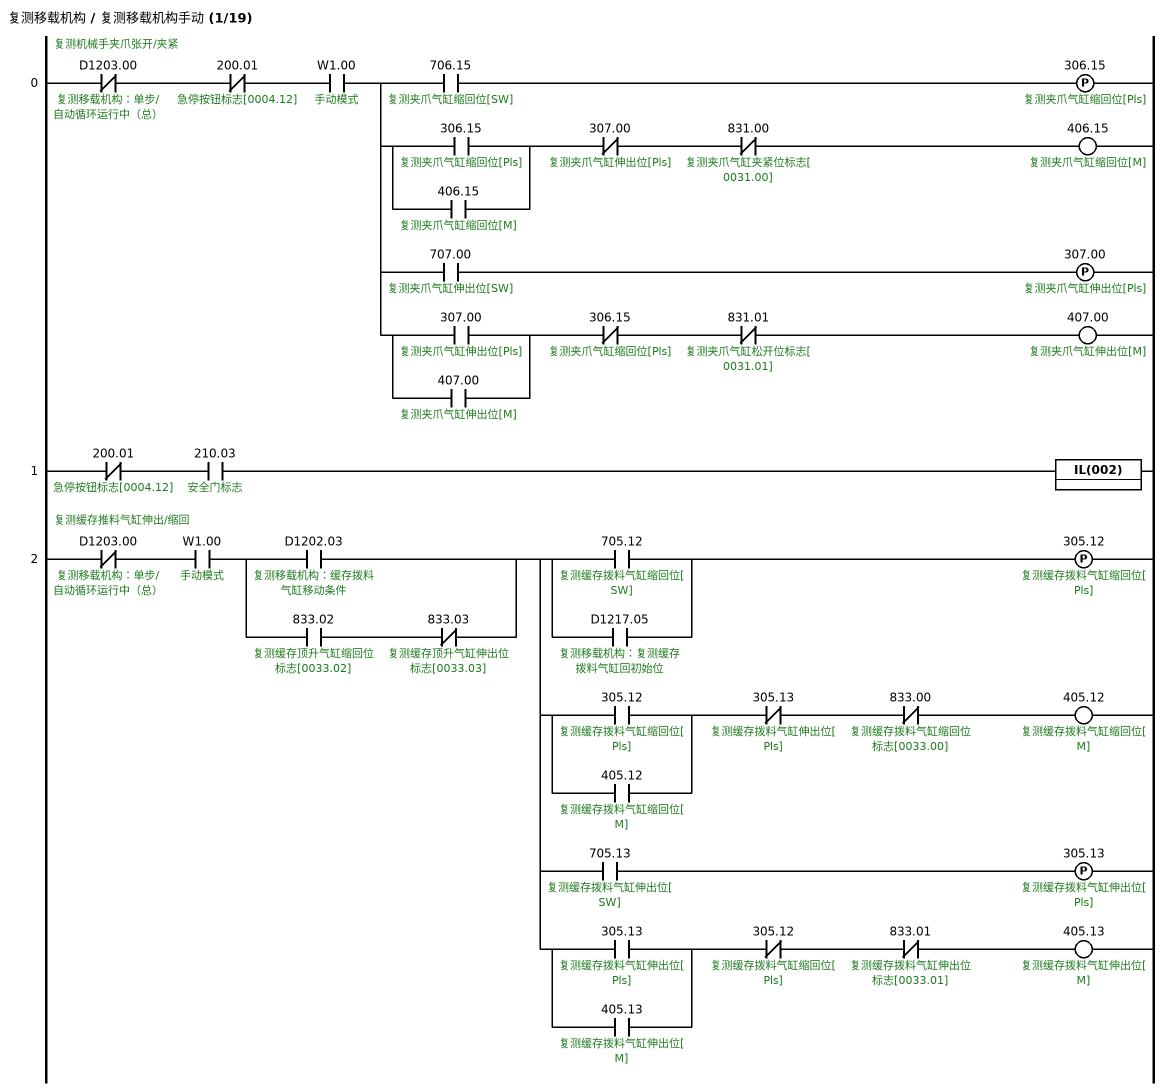
; [picture p552: 复测移载机构 / 复测移载机构手动, rungs 0-2]
; rung 0: 复测机械手夹爪张开/夹紧
LDNOT D1203.00  ; 复测移载机构：单步/自动循环运行中（总）
ANDNOT 200.01  ; 急停按钮标志[0004.12]
AND W1.00  ; 手动模式
OUT TR0
AND 706.15  ; 复测夹爪气缸缩回位[SW]
DIFU(013) 306.15  ; 复测夹爪气缸缩回位[Pls]
LD TR0
LD 306.15  ; 复测夹爪气缸缩回位[Pls]
OR 406.15  ; 复测夹爪气缸缩回位[M]
ANDLD
ANDNOT 307.00  ; 复测夹爪气缸伸出位[Pls]
ANDNOT 831.00  ; 复测夹爪气缸夹紧位标志[0031.00]
OUT 406.15  ; 复测夹爪气缸缩回位[M]
LD TR0
AND 707.00  ; 复测夹爪气缸伸出位[SW]
DIFU(013) 307.00  ; 复测夹爪气缸伸出位[Pls]
LD TR0
LD 307.00  ; 复测夹爪气缸伸出位[Pls]
OR 407.00  ; 复测夹爪气缸伸出位[M]
ANDLD
ANDNOT 306.15  ; 复测夹爪气缸缩回位[Pls]
ANDNOT 831.01  ; 复测夹爪气缸松开位标志[0031.01]
OUT 407.00  ; 复测夹爪气缸伸出位[M]
; rung 1
LDNOT 200.01  ; 急停按钮标志[0004.12]
AND 210.03  ; 安全门标志
IL(002)
; rung 2: 复测缓存推料气缸伸出/缩回
LDNOT D1203.00  ; 复测移载机构：单步/自动循环运行中（总）
AND W1.00  ; 手动模式
LD D1202.03  ; 复测移载机构：缓存拨料气缸移动条件
LD 833.02  ; 复测缓存顶升气缸缩回位标志[0033.02]
ANDNOT 833.03  ; 复测缓存顶升气缸伸出位标志[0033.03]
ORLD
ANDLD
OUT TR0
LD 705.12  ; 复测缓存拨料气缸缩回位[SW]
OR D1217.05  ; 复测移载机构：复测缓存拨料气缸回初始位
ANDLD
DIFU(013) 305.12  ; 复测缓存拨料气缸缩回位[Pls]
LD TR0
LD 305.12  ; 复测缓存拨料气缸缩回位[Pls]
OR 405.12  ; 复测缓存拨料气缸缩回位[M]
ANDLD
ANDNOT 305.13  ; 复测缓存拨料气缸伸出位[Pls]
ANDNOT 833.00  ; 复测缓存拨料气缸缩回位标志[0033.00]
OUT 405.12  ; 复测缓存拨料气缸缩回位[M]
LD TR0
AND 705.13  ; 复测缓存拨料气缸伸出位[SW]
DIFU(013) 305.13  ; 复测缓存拨料气缸伸出位[Pls]
LD TR0
LD 305.13  ; 复测缓存拨料气缸伸出位[Pls]
OR 405.13  ; 复测缓存拨料气缸伸出位[M]
ANDLD
ANDNOT 305.12  ; 复测缓存拨料气缸缩回位[Pls]
ANDNOT 833.01  ; 复测缓存拨料气缸伸出位标志[0033.01]
OUT 405.13  ; 复测缓存拨料气缸伸出位[M]

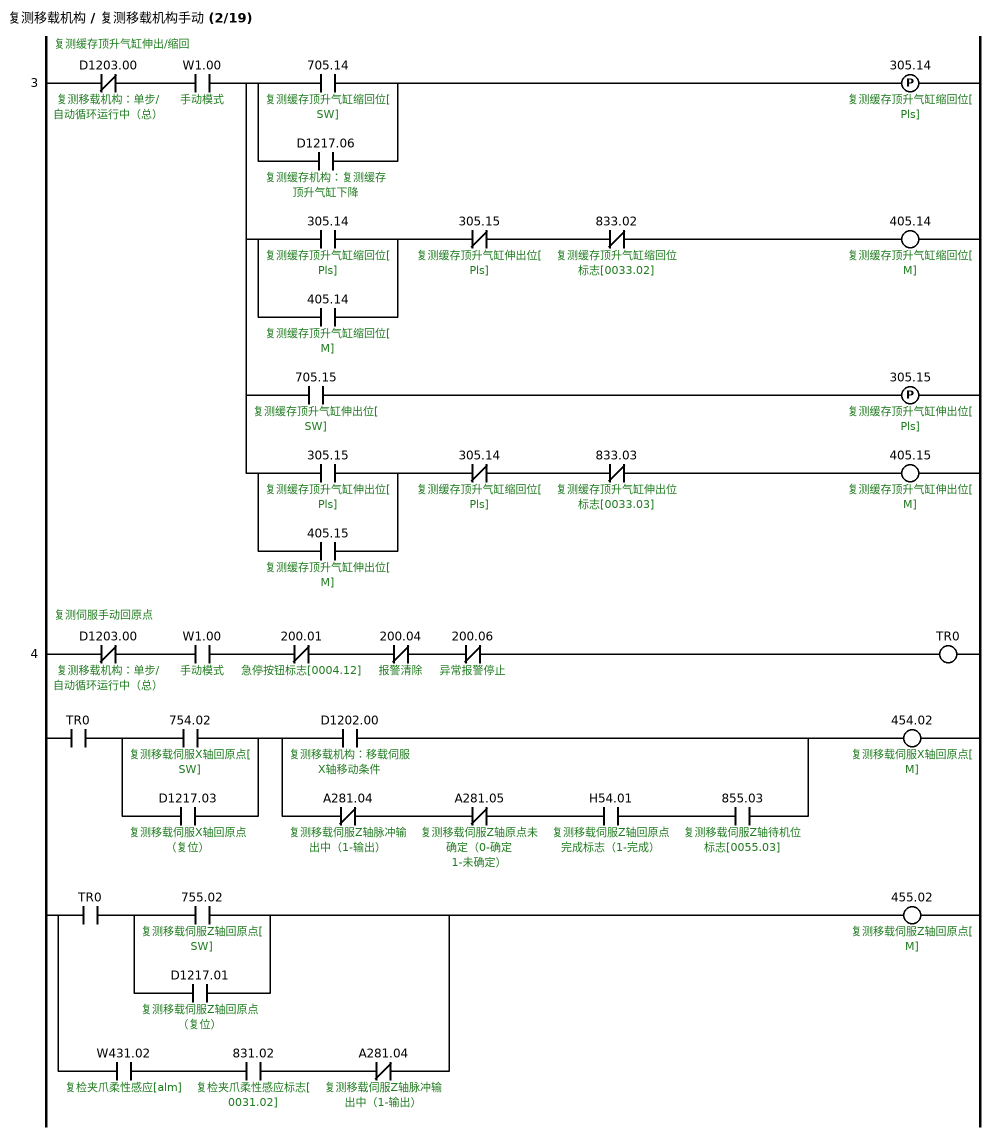
; rung 3: 复测缓存顶升气缸伸出/缩回
LDNOT D1203.00  ; 复测移载机构：单步/自动循环运行中（总）
AND W1.00  ; 手动模式
OUT TR0
LD 705.14  ; 复测缓存顶升气缸缩回位[SW]
OR D1217.06  ; 复测缓存机构：复测缓存顶升气缸下降
ANDLD
DIFU(013) 305.14  ; 复测缓存顶升气缸缩回位[Pls]
LD TR0
LD 305.14  ; 复测缓存顶升气缸缩回位[Pls]
OR 405.14  ; 复测缓存顶升气缸缩回位[M]
ANDLD
ANDNOT 305.15  ; 复测缓存顶升气缸伸出位[Pls]
ANDNOT 833.02  ; 复测缓存顶升气缸缩回位标志[0033.02]
OUT 405.14  ; 复测缓存顶升气缸缩回位[M]
LD TR0
AND 705.15  ; 复测缓存顶升气缸伸出位[SW]
DIFU(013) 305.15  ; 复测缓存顶升气缸伸出位[Pls]
LD TR0
LD 305.15  ; 复测缓存顶升气缸伸出位[Pls]
OR 405.15  ; 复测缓存顶升气缸伸出位[M]
ANDLD
ANDNOT 305.14  ; 复测缓存顶升气缸缩回位[Pls]
ANDNOT 833.03  ; 复测缓存顶升气缸伸出位标志[0033.03]
OUT 405.15  ; 复测缓存顶升气缸伸出位[M]
; rung 4: 复测伺服手动回原点
LDNOT D1203.00  ; 复测移载机构：单步/自动循环运行中（总）
AND W1.00  ; 手动模式
ANDNOT 200.01  ; 急停按钮标志[0004.12]
ANDNOT 200.04  ; 报警清除
ANDNOT 200.06  ; 异常报警停止
OUT TR0
LD 754.02  ; 复测移载伺服X轴回原点[SW]
OR D1217.03  ; 复测移载伺服X轴回原点（复位）
ANDLD
LD D1202.00  ; 复测移载机构：移载伺服X轴移动条件
LDNOT A281.04  ; 复测移载伺服Z轴脉冲输出中（1-输出）
ANDNOT A281.05  ; 复测移载伺服Z轴原点未确定（0-确定  1-未确定）
AND H54.01  ; 复测移载伺服Z轴回原点完成标志（1-完成）
AND 855.03  ; 复测移载伺服Z轴待机位标志[0055.03]
ORLD
ANDLD
OUT 454.02  ; 复测移载伺服X轴回原点[M]
LD TR0
LD 755.02  ; 复测移载伺服Z轴回原点[SW]
OR D1217.01  ; 复测移载伺服Z轴回原点（复位）
ANDLD
LD W431.02  ; 复检夹爪柔性感应[alm]
AND 831.02  ; 复检夹爪柔性感应标志[0031.02]
ANDNOT A281.04  ; 复测移载伺服Z轴脉冲输出中（1-输出）
ORLD
OUT 455.02  ; 复测移载伺服Z轴回原点[M]

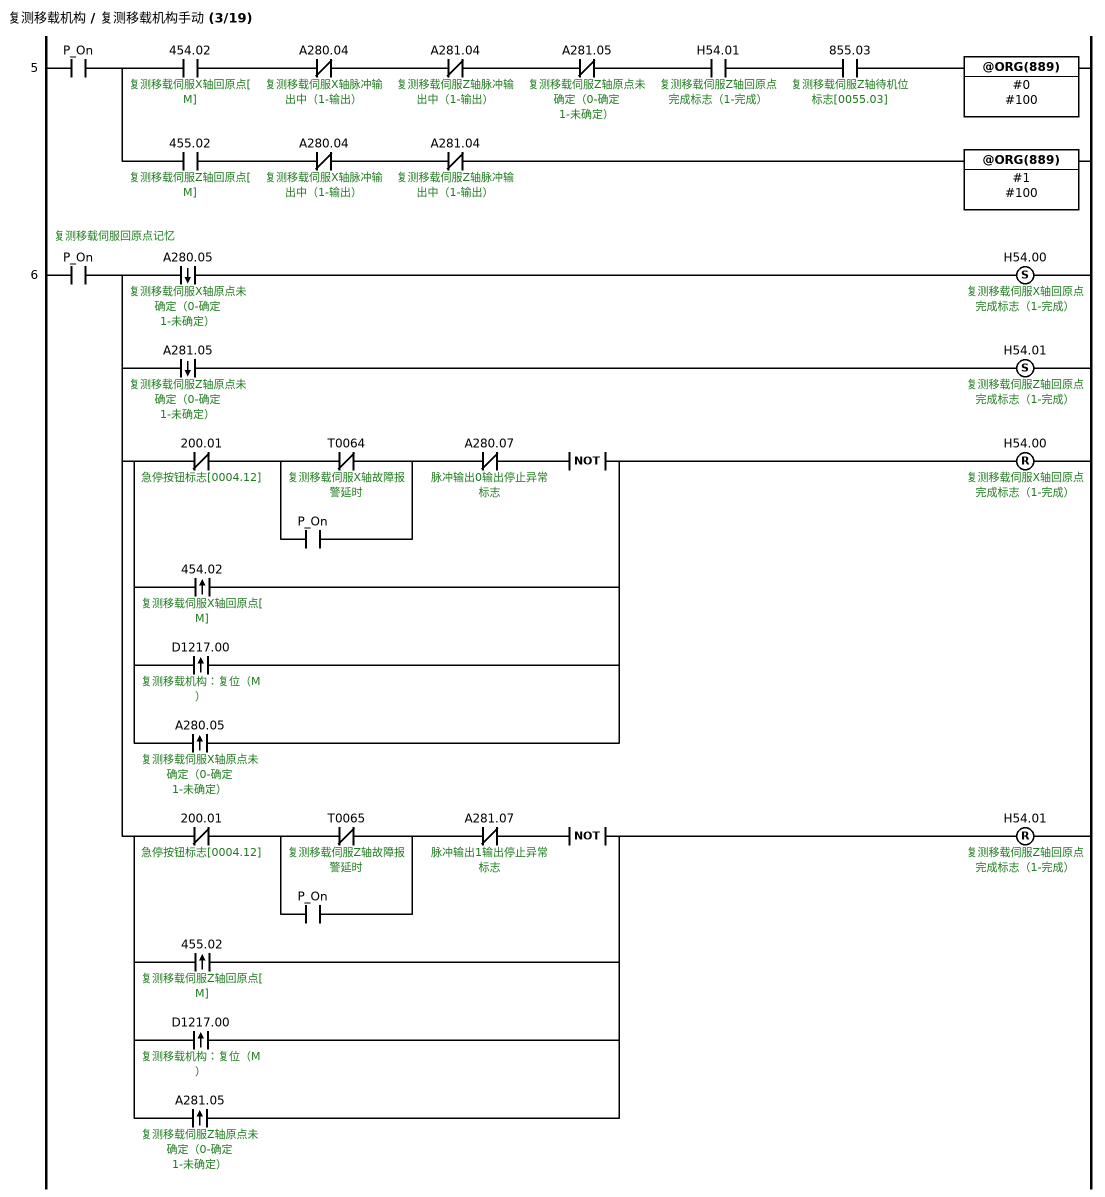
; rung 5
LD P_On
OUT TR0
AND 454.02  ; 复测移载伺服X轴回原点[M]
ANDNOT A280.04  ; 复测移载伺服X轴脉冲输出中（1-输出）
ANDNOT A281.04  ; 复测移载伺服Z轴脉冲输出中（1-输出）
ANDNOT A281.05  ; 复测移载伺服Z轴原点未确定（0-确定  1-未确定）
AND H54.01  ; 复测移载伺服Z轴回原点完成标志（1-完成）
AND 855.03  ; 复测移载伺服Z轴待机位标志[0055.03]
@ORG(889) #0 #100
LD TR0
AND 455.02  ; 复测移载伺服Z轴回原点[M]
ANDNOT A280.04  ; 复测移载伺服X轴脉冲输出中（1-输出）
ANDNOT A281.04  ; 复测移载伺服Z轴脉冲输出中（1-输出）
@ORG(889) #1 #100
; rung 6: 复测移载伺服回原点记忆
LD P_On
OUT TR0
%AND A280.05  ; 复测移载伺服X轴原点未确定（0-确定  1-未确定）
SET H54.00  ; 复测移载伺服X轴回原点完成标志（1-完成）
LD TR0
%AND A281.05  ; 复测移载伺服Z轴原点未确定（0-确定  1-未确定）
SET H54.01  ; 复测移载伺服Z轴回原点完成标志（1-完成）
LD TR0
LDNOT 200.01  ; 急停按钮标志[0004.12]
LDNOT T0064  ; 复测移载伺服X轴故障报警延时
OR P_On
ANDLD
ANDNOT A280.07  ; 脉冲输出0输出停止异常标志
NOT(520)
@OR 454.02  ; 复测移载伺服X轴回原点[M]
@OR D1217.00  ; 复测移载机构：复位（M）
@OR A280.05  ; 复测移载伺服X轴原点未确定（0-确定  1-未确定）
ANDLD
RSET H54.00  ; 复测移载伺服X轴回原点完成标志（1-完成）
LD TR0
LDNOT 200.01  ; 急停按钮标志[0004.12]
LDNOT T0065  ; 复测移载伺服Z轴故障报警延时
OR P_On
ANDLD
ANDNOT A281.07  ; 脉冲输出1输出停止异常标志
NOT(520)
@OR 455.02  ; 复测移载伺服Z轴回原点[M]
@OR D1217.00  ; 复测移载机构：复位（M）
@OR A281.05  ; 复测移载伺服Z轴原点未确定（0-确定  1-未确定）
ANDLD
RSET H54.01  ; 复测移载伺服Z轴回原点完成标志（1-完成）

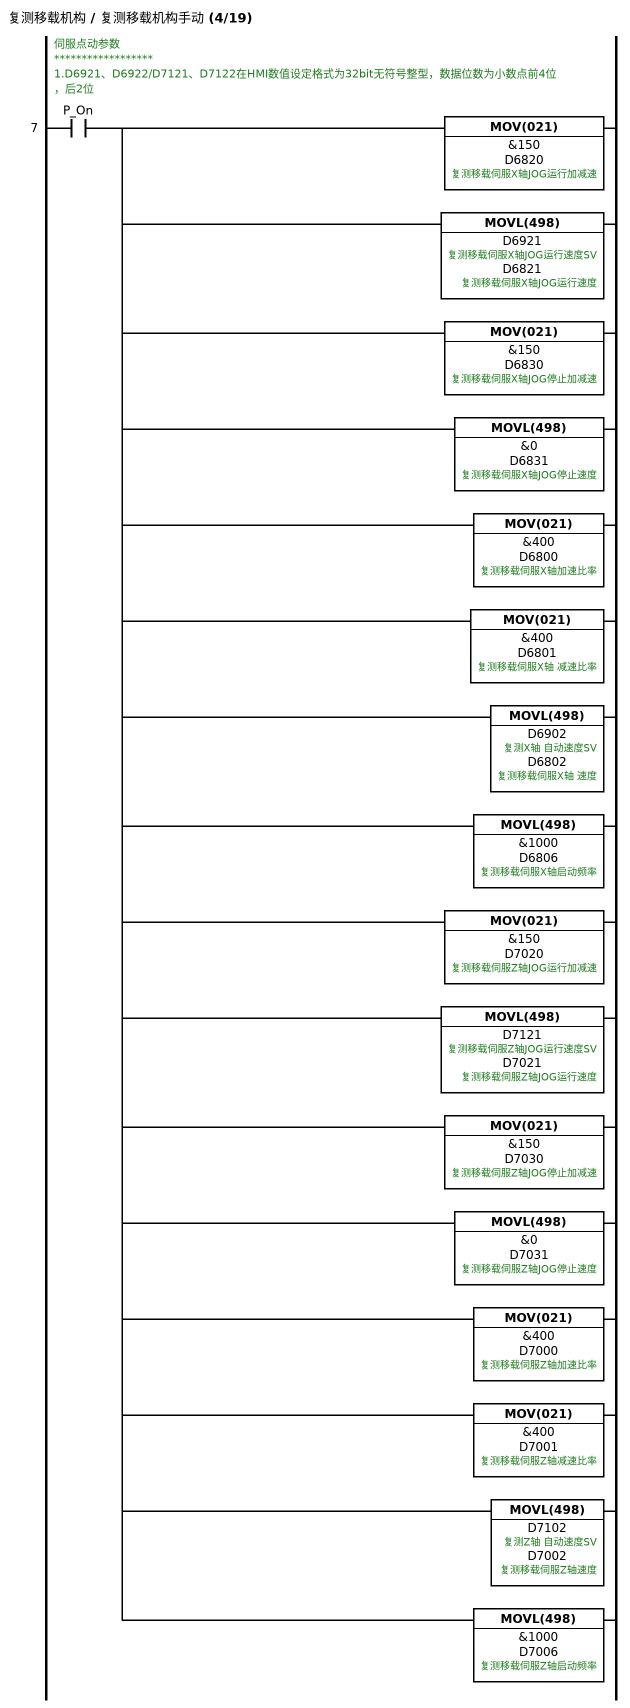
; rung 7: 伺服点动参数 / ****************** / 1.D6921、D6922/D7121、D7122在HMI数值设定格式为32bit无符号整型，数据位数为小数点前4位，后2位
LD P_On
MOV(021) &150 D6820  ; 复测移载伺服X轴JOG运行加减速
MOVL(498) D6921 D6821  ; 复测移载伺服X轴JOG运行速度SV, 复测移载伺服X轴JOG运行速度
MOV(021) &150 D6830  ; 复测移载伺服X轴JOG停止加减速
MOVL(498) &0 D6831  ; 复测移载伺服X轴JOG停止速度
MOV(021) &400 D6800  ; 复测移载伺服X轴加速比率
MOV(021) &400 D6801  ; 复测移载伺服X轴 减速比率
MOVL(498) D6902 D6802  ; 复测X轴 自动速度SV, 复测移载伺服X轴 速度
MOVL(498) &1000 D6806  ; 复测移载伺服X轴启动频率
MOV(021) &150 D7020  ; 复测移载伺服Z轴JOG运行加减速
MOVL(498) D7121 D7021  ; 复测移载伺服Z轴JOG运行速度SV, 复测移载伺服Z轴JOG运行速度
MOV(021) &150 D7030  ; 复测移载伺服Z轴JOG停止加减速
MOVL(498) &0 D7031  ; 复测移载伺服Z轴JOG停止速度
MOV(021) &400 D7000  ; 复测移载伺服Z轴加速比率
MOV(021) &400 D7001  ; 复测移载伺服Z轴减速比率
MOVL(498) D7102 D7002  ; 复测Z轴 自动速度SV, 复测移载伺服Z轴速度
MOVL(498) &1000 D7006  ; 复测移载伺服Z轴启动频率

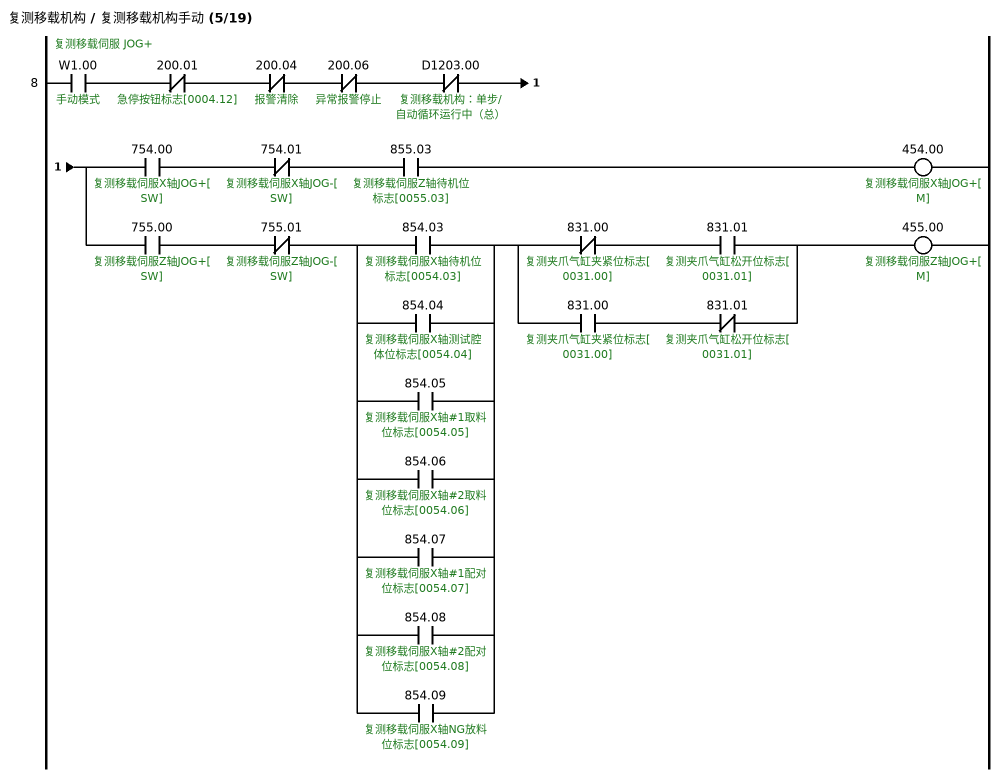
; rung 8: 复测移载伺服 JOG+
LD W1.00  ; 手动模式
ANDNOT 200.01  ; 急停按钮标志[0004.12]
ANDNOT 200.04  ; 报警清除
ANDNOT 200.06  ; 异常报警停止
ANDNOT D1203.00  ; 复测移载机构：单步/自动循环运行中（总）
OUT TR0
AND 754.00  ; 复测移载伺服X轴JOG+[SW]
ANDNOT 754.01  ; 复测移载伺服X轴JOG-[SW]
AND 855.03  ; 复测移载伺服Z轴待机位标志[0055.03]
OUT 454.00  ; 复测移载伺服X轴JOG+[M]
LD TR0
AND 755.00  ; 复测移载伺服Z轴JOG+[SW]
ANDNOT 755.01  ; 复测移载伺服Z轴JOG-[SW]
LD 854.03  ; 复测移载伺服X轴待机位标志[0054.03]
OR 854.04  ; 复测移载伺服X轴测试腔体位标志[0054.04]
OR 854.05  ; 复测移载伺服X轴#1取料位标志[0054.05]
OR 854.06  ; 复测移载伺服X轴#2取料位标志[0054.06]
OR 854.07  ; 复测移载伺服X轴#1配对位标志[0054.07]
OR 854.08  ; 复测移载伺服X轴#2配对位标志[0054.08]
OR 854.09  ; 复测移载伺服X轴NG放料位标志[0054.09]
ANDLD
LDNOT 831.00  ; 复测夹爪气缸夹紧位标志[0031.00]
AND 831.01  ; 复测夹爪气缸松开位标志[0031.01]
LD 831.00  ; 复测夹爪气缸夹紧位标志[0031.00]
ANDNOT 831.01  ; 复测夹爪气缸松开位标志[0031.01]
ORLD
ANDLD
OUT 455.00  ; 复测移载伺服Z轴JOG+[M]

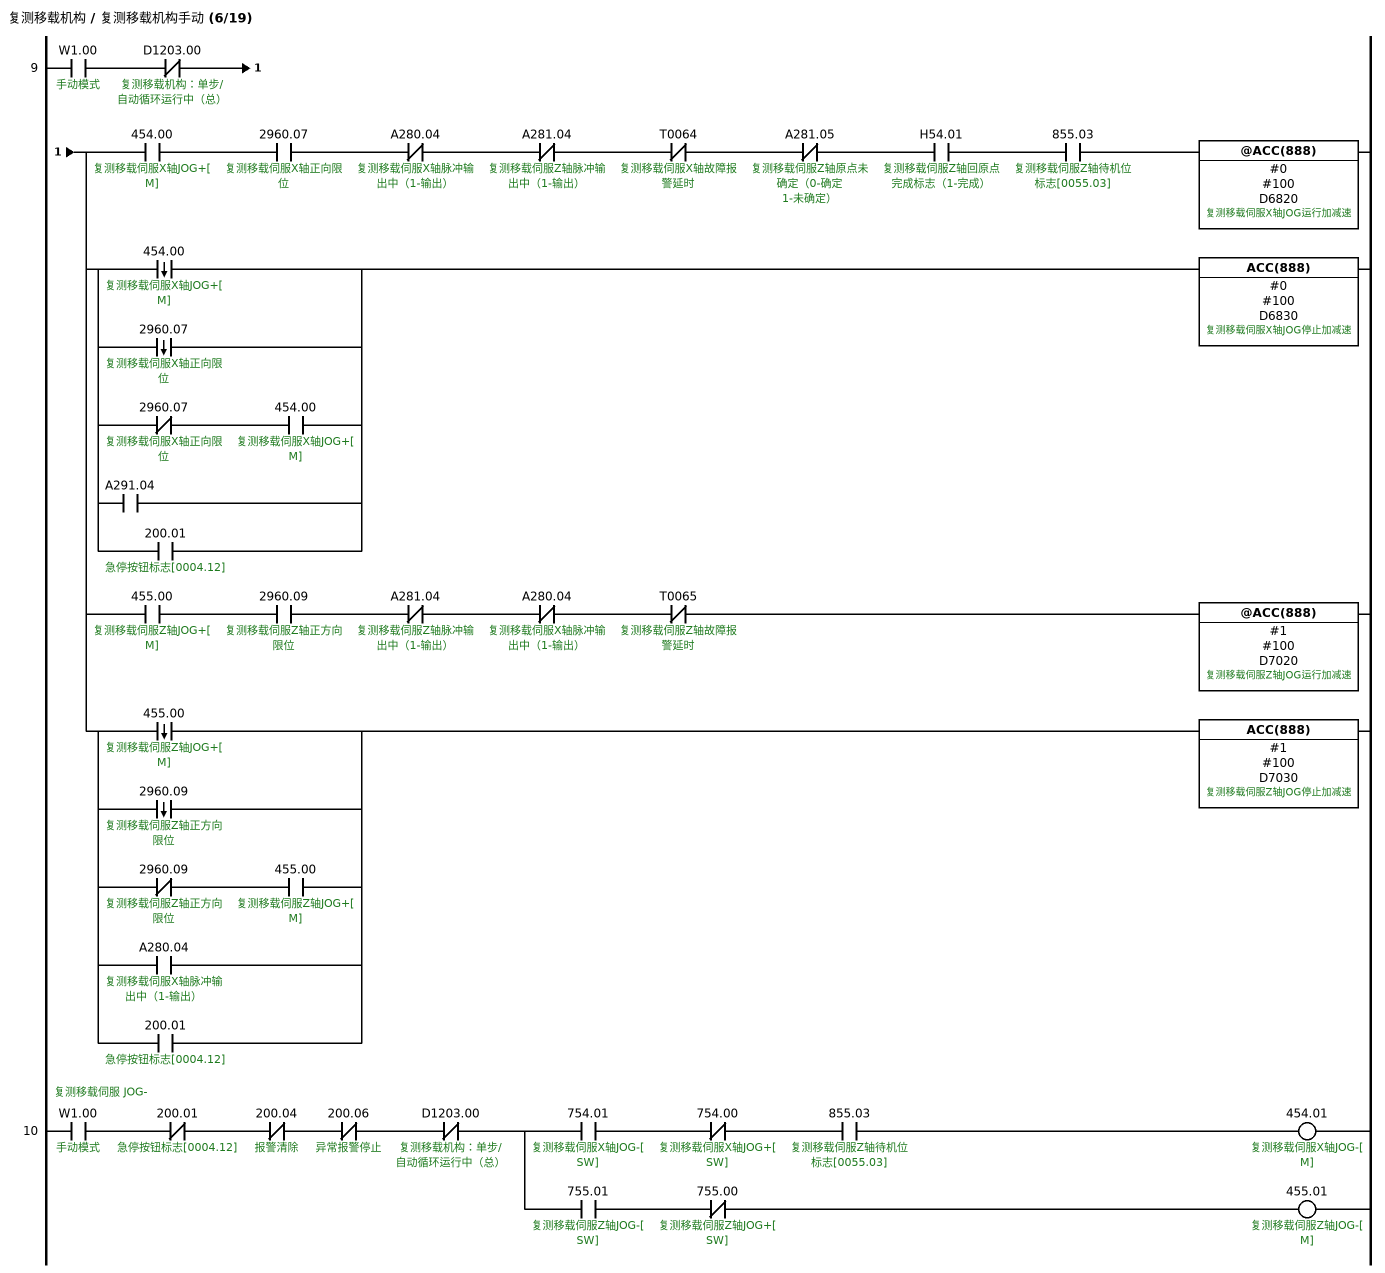
; rung 9
LD W1.00  ; 手动模式
ANDNOT D1203.00  ; 复测移载机构：单步/自动循环运行中（总）
OUT TR0
AND 454.00  ; 复测移载伺服X轴JOG+[M]
AND 2960.07  ; 复测移载伺服X轴正向限位
ANDNOT A280.04  ; 复测移载伺服X轴脉冲输出中（1-输出）
ANDNOT A281.04  ; 复测移载伺服Z轴脉冲输出中（1-输出）
ANDNOT T0064  ; 复测移载伺服X轴故障报警延时
ANDNOT A281.05  ; 复测移载伺服Z轴原点未确定（0-确定  1-未确定）
AND H54.01  ; 复测移载伺服Z轴回原点完成标志（1-完成）
AND 855.03  ; 复测移载伺服Z轴待机位标志[0055.03]
@ACC(888) #0 #100 D6820  ; 复测移载伺服X轴JOG运行加减速
LD TR0
%LD 454.00  ; 复测移载伺服X轴JOG+[M]
%OR 2960.07  ; 复测移载伺服X轴正向限位
LDNOT 2960.07  ; 复测移载伺服X轴正向限位
AND 454.00  ; 复测移载伺服X轴JOG+[M]
ORLD
OR A291.04
OR 200.01  ; 急停按钮标志[0004.12]
ANDLD
ACC(888) #0 #100 D6830  ; 复测移载伺服X轴JOG停止加减速
LD TR0
AND 455.00  ; 复测移载伺服Z轴JOG+[M]
AND 2960.09  ; 复测移载伺服Z轴正方向限位
ANDNOT A281.04  ; 复测移载伺服Z轴脉冲输出中（1-输出）
ANDNOT A280.04  ; 复测移载伺服X轴脉冲输出中（1-输出）
ANDNOT T0065  ; 复测移载伺服Z轴故障报警延时
@ACC(888) #1 #100 D7020  ; 复测移载伺服Z轴JOG运行加减速
LD TR0
%LD 455.00  ; 复测移载伺服Z轴JOG+[M]
%OR 2960.09  ; 复测移载伺服Z轴正方向限位
LDNOT 2960.09  ; 复测移载伺服Z轴正方向限位
AND 455.00  ; 复测移载伺服Z轴JOG+[M]
ORLD
OR A280.04  ; 复测移载伺服X轴脉冲输出中（1-输出）
OR 200.01  ; 急停按钮标志[0004.12]
ANDLD
ACC(888) #1 #100 D7030  ; 复测移载伺服Z轴JOG停止加减速
; rung 10: 复测移载伺服 JOG-
LD W1.00  ; 手动模式
ANDNOT 200.01  ; 急停按钮标志[0004.12]
ANDNOT 200.04  ; 报警清除
ANDNOT 200.06  ; 异常报警停止
ANDNOT D1203.00  ; 复测移载机构：单步/自动循环运行中（总）
OUT TR0
AND 754.01  ; 复测移载伺服X轴JOG-[SW]
ANDNOT 754.00  ; 复测移载伺服X轴JOG+[SW]
AND 855.03  ; 复测移载伺服Z轴待机位标志[0055.03]
OUT 454.01  ; 复测移载伺服X轴JOG-[M]
LD TR0
AND 755.01  ; 复测移载伺服Z轴JOG-[SW]
ANDNOT 755.00  ; 复测移载伺服Z轴JOG+[SW]
OUT 455.01  ; 复测移载伺服Z轴JOG-[M]

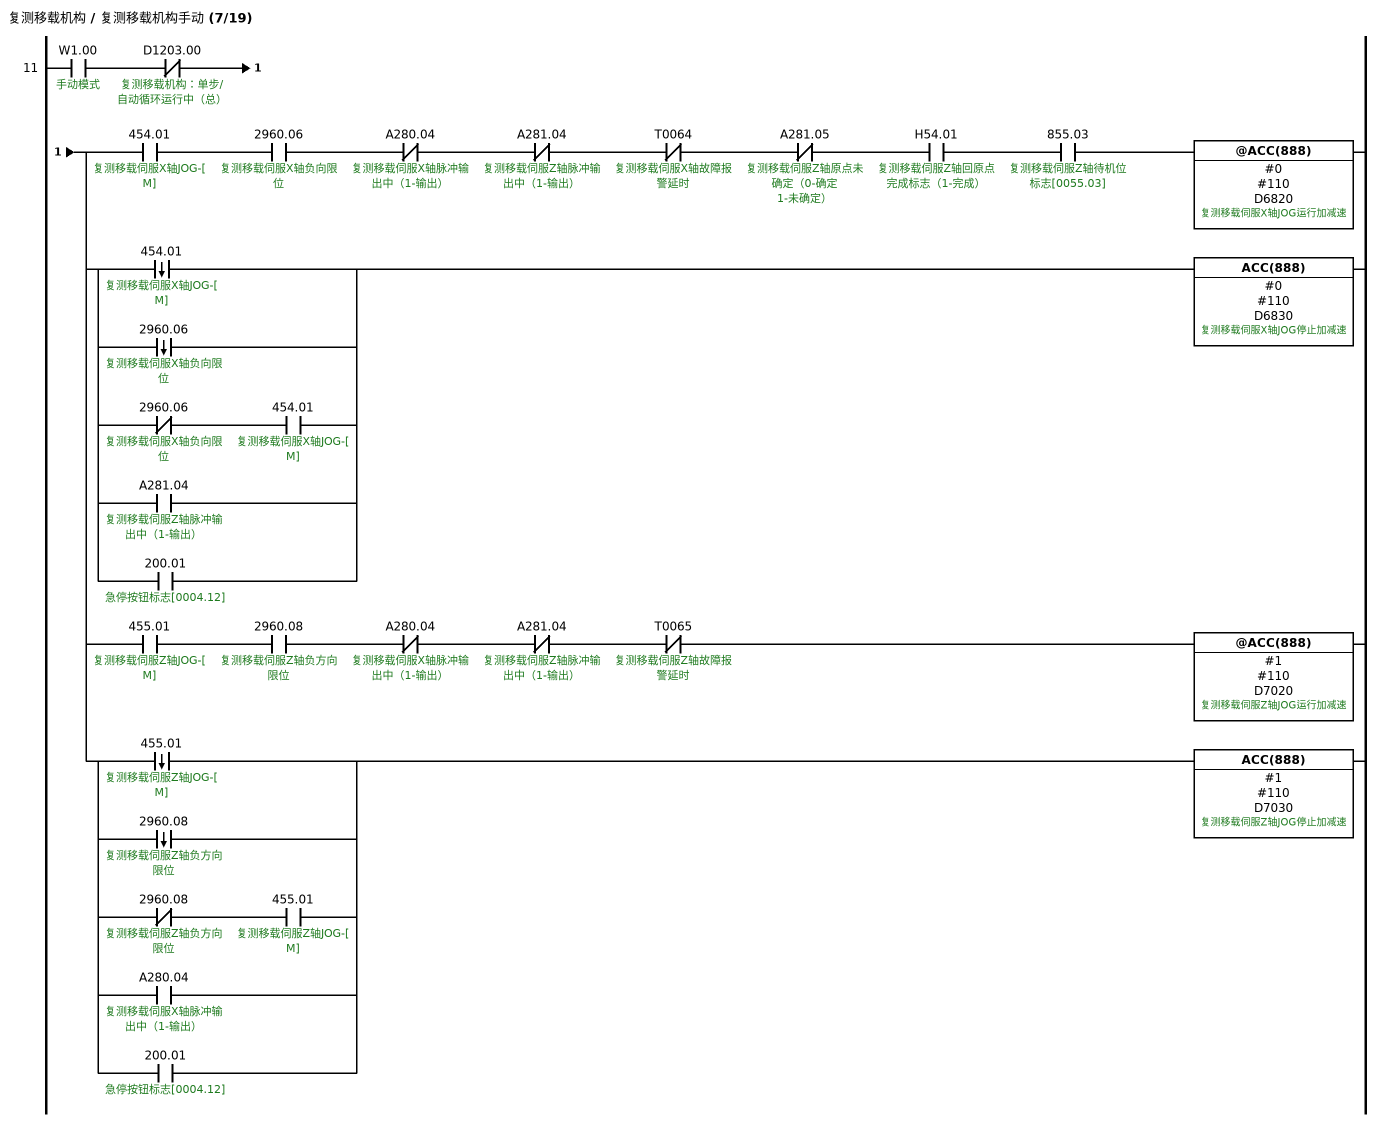
; rung 11
LD W1.00  ; 手动模式
ANDNOT D1203.00  ; 复测移载机构：单步/自动循环运行中（总）
OUT TR0
AND 454.01  ; 复测移载伺服X轴JOG-[M]
AND 2960.06  ; 复测移载伺服X轴负向限位
ANDNOT A280.04  ; 复测移载伺服X轴脉冲输出中（1-输出）
ANDNOT A281.04  ; 复测移载伺服Z轴脉冲输出中（1-输出）
ANDNOT T0064  ; 复测移载伺服X轴故障报警延时
ANDNOT A281.05  ; 复测移载伺服Z轴原点未确定（0-确定  1-未确定）
AND H54.01  ; 复测移载伺服Z轴回原点完成标志（1-完成）
AND 855.03  ; 复测移载伺服Z轴待机位标志[0055.03]
@ACC(888) #0 #110 D6820  ; 复测移载伺服X轴JOG运行加减速
LD TR0
%LD 454.01  ; 复测移载伺服X轴JOG-[M]
%OR 2960.06  ; 复测移载伺服X轴负向限位
LDNOT 2960.06  ; 复测移载伺服X轴负向限位
AND 454.01  ; 复测移载伺服X轴JOG-[M]
ORLD
OR A281.04  ; 复测移载伺服Z轴脉冲输出中（1-输出）
OR 200.01  ; 急停按钮标志[0004.12]
ANDLD
ACC(888) #0 #110 D6830  ; 复测移载伺服X轴JOG停止加减速
LD TR0
AND 455.01  ; 复测移载伺服Z轴JOG-[M]
AND 2960.08  ; 复测移载伺服Z轴负方向限位
ANDNOT A280.04  ; 复测移载伺服X轴脉冲输出中（1-输出）
ANDNOT A281.04  ; 复测移载伺服Z轴脉冲输出中（1-输出）
ANDNOT T0065  ; 复测移载伺服Z轴故障报警延时
@ACC(888) #1 #110 D7020  ; 复测移载伺服Z轴JOG运行加减速
LD TR0
%LD 455.01  ; 复测移载伺服Z轴JOG-[M]
%OR 2960.08  ; 复测移载伺服Z轴负方向限位
LDNOT 2960.08  ; 复测移载伺服Z轴负方向限位
AND 455.01  ; 复测移载伺服Z轴JOG-[M]
ORLD
OR A280.04  ; 复测移载伺服X轴脉冲输出中（1-输出）
OR 200.01  ; 急停按钮标志[0004.12]
ANDLD
ACC(888) #1 #110 D7030  ; 复测移载伺服Z轴JOG停止加减速

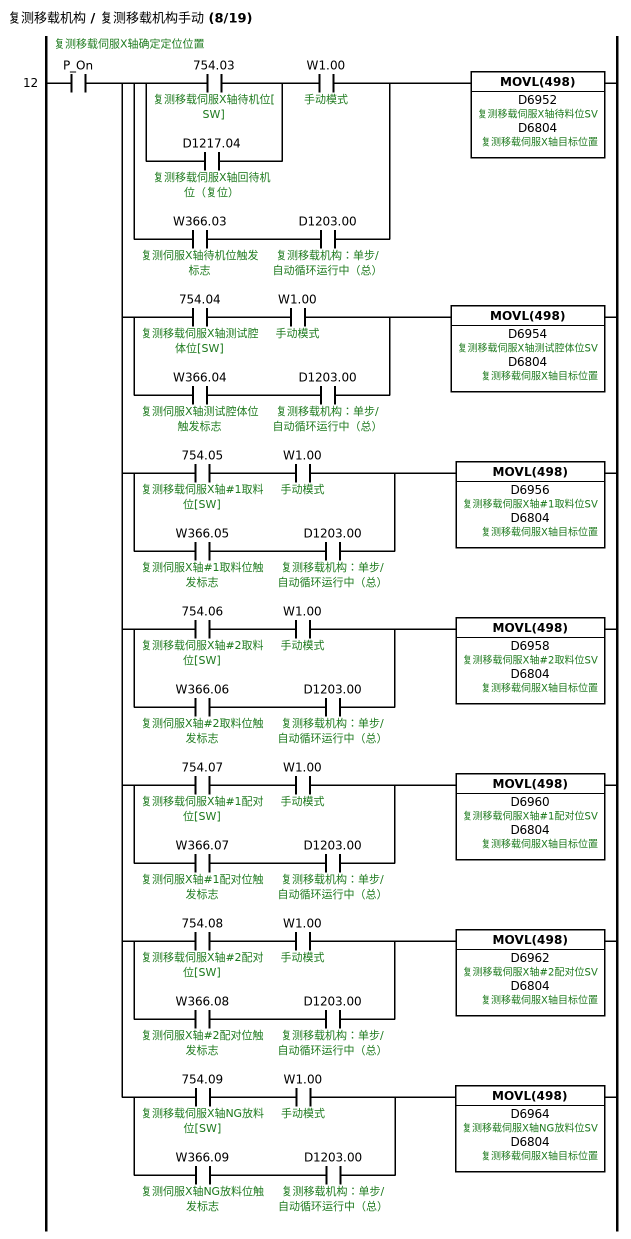
; rung 12: 复测移载伺服X轴确定定位位置
LD P_On
OUT TR0
LD 754.03  ; 复测移载伺服X轴待机位[SW]
OR D1217.04  ; 复测移载伺服X轴回待机位（复位）
AND W1.00  ; 手动模式
LD W366.03  ; 复测伺服X轴待机位触发标志
AND D1203.00  ; 复测移载机构：单步/自动循环运行中（总）
ORLD
ANDLD
MOVL(498) D6952 D6804  ; 复测移载伺服X轴待料位SV, 复测移载伺服X轴目标位置
LD TR0
LD 754.04  ; 复测移载伺服X轴测试腔体位[SW]
AND W1.00  ; 手动模式
LD W366.04  ; 复测伺服X轴测试腔体位触发标志
AND D1203.00  ; 复测移载机构：单步/自动循环运行中（总）
ORLD
ANDLD
MOVL(498) D6954 D6804  ; 复测移载伺服X轴测试腔体位SV, 复测移载伺服X轴目标位置
LD TR0
LD 754.05  ; 复测移载伺服X轴#1取料位[SW]
AND W1.00  ; 手动模式
LD W366.05  ; 复测伺服X轴#1取料位触发标志
AND D1203.00  ; 复测移载机构：单步/自动循环运行中（总）
ORLD
ANDLD
MOVL(498) D6956 D6804  ; 复测移载伺服X轴#1取料位SV, 复测移载伺服X轴目标位置
LD TR0
LD 754.06  ; 复测移载伺服X轴#2取料位[SW]
AND W1.00  ; 手动模式
LD W366.06  ; 复测伺服X轴#2取料位触发标志
AND D1203.00  ; 复测移载机构：单步/自动循环运行中（总）
ORLD
ANDLD
MOVL(498) D6958 D6804  ; 复测移载伺服X轴#2取料位SV, 复测移载伺服X轴目标位置
LD TR0
LD 754.07  ; 复测移载伺服X轴#1配对位[SW]
AND W1.00  ; 手动模式
LD W366.07  ; 复测伺服X轴#1配对位触发标志
AND D1203.00  ; 复测移载机构：单步/自动循环运行中（总）
ORLD
ANDLD
MOVL(498) D6960 D6804  ; 复测移载伺服X轴#1配对位SV, 复测移载伺服X轴目标位置
LD TR0
LD 754.08  ; 复测移载伺服X轴#2配对位[SW]
AND W1.00  ; 手动模式
LD W366.08  ; 复测伺服X轴#2配对位触发标志
AND D1203.00  ; 复测移载机构：单步/自动循环运行中（总）
ORLD
ANDLD
MOVL(498) D6962 D6804  ; 复测移载伺服X轴#2配对位SV, 复测移载伺服X轴目标位置
LD TR0
LD 754.09  ; 复测移载伺服X轴NG放料位[SW]
AND W1.00  ; 手动模式
LD W366.09  ; 复测伺服X轴NG放料位触发标志
AND D1203.00  ; 复测移载机构：单步/自动循环运行中（总）
ORLD
ANDLD
MOVL(498) D6964 D6804  ; 复测移载伺服X轴NG放料位SV, 复测移载伺服X轴目标位置

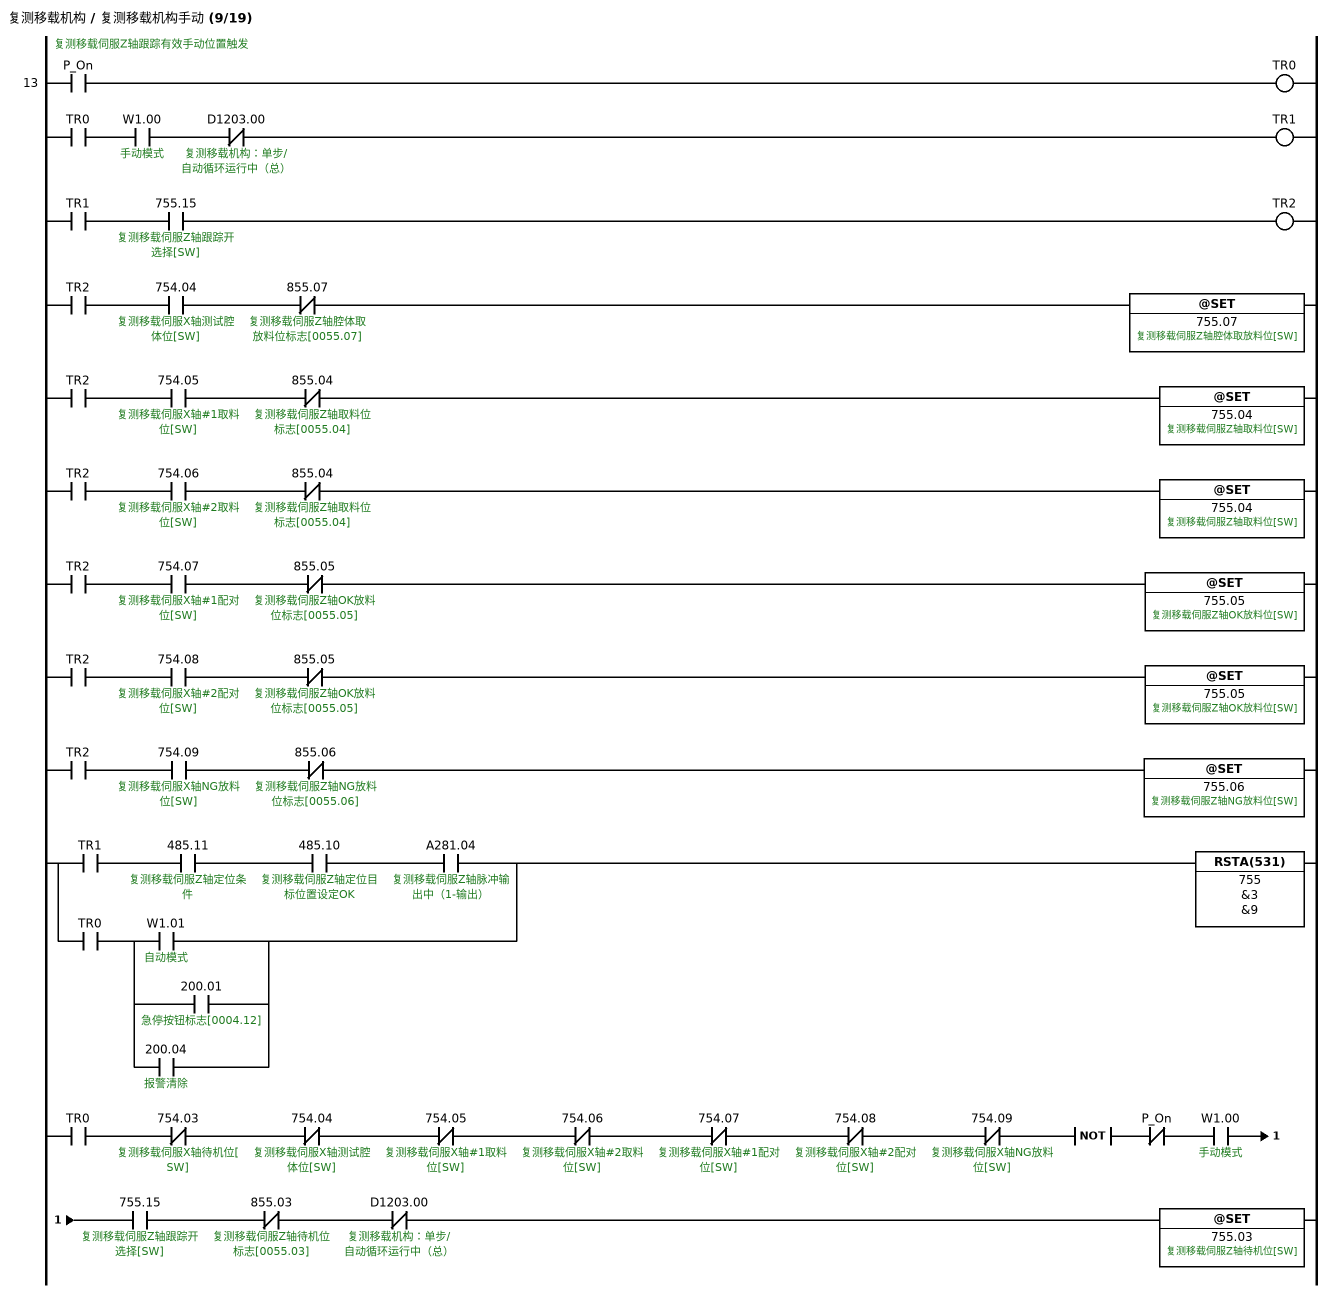
; rung 13: 复测移载伺服Z轴跟踪有效手动位置触发
LD P_On
OUT TR0
AND W1.00  ; 手动模式
ANDNOT D1203.00  ; 复测移载机构：单步/自动循环运行中（总）
OUT TR1
AND 755.15  ; 复测移载伺服Z轴跟踪开选择[SW]
OUT TR2
AND 754.04  ; 复测移载伺服X轴测试腔体位[SW]
ANDNOT 855.07  ; 复测移载伺服Z轴腔体取放料位标志[0055.07]
@SET 755.07  ; 复测移载伺服Z轴腔体取放料位[SW]
LD TR2
AND 754.05  ; 复测移载伺服X轴#1取料位[SW]
ANDNOT 855.04  ; 复测移载伺服Z轴取料位标志[0055.04]
@SET 755.04  ; 复测移载伺服Z轴取料位[SW]
LD TR2
AND 754.06  ; 复测移载伺服X轴#2取料位[SW]
ANDNOT 855.04  ; 复测移载伺服Z轴取料位标志[0055.04]
@SET 755.04  ; 复测移载伺服Z轴取料位[SW]
LD TR2
AND 754.07  ; 复测移载伺服X轴#1配对位[SW]
ANDNOT 855.05  ; 复测移载伺服Z轴OK放料位标志[0055.05]
@SET 755.05  ; 复测移载伺服Z轴OK放料位[SW]
LD TR2
AND 754.08  ; 复测移载伺服X轴#2配对位[SW]
ANDNOT 855.05  ; 复测移载伺服Z轴OK放料位标志[0055.05]
@SET 755.05  ; 复测移载伺服Z轴OK放料位[SW]
LD TR2
AND 754.09  ; 复测移载伺服X轴NG放料位[SW]
ANDNOT 855.06  ; 复测移载伺服Z轴NG放料位标志[0055.06]
@SET 755.06  ; 复测移载伺服Z轴NG放料位[SW]
LD TR1
AND 485.11  ; 复测移载伺服Z轴定位条件
AND 485.10  ; 复测移载伺服Z轴定位目标位置设定OK
AND A281.04  ; 复测移载伺服Z轴脉冲输出中（1-输出）
LD TR0
LD W1.01  ; 自动模式
OR 200.01  ; 急停按钮标志[0004.12]
OR 200.04  ; 报警清除
ANDLD
ORLD
RSTA(531) 755 &3 &9
LD TR0
ANDNOT 754.03  ; 复测移载伺服X轴待机位[SW]
ANDNOT 754.04  ; 复测移载伺服X轴测试腔体位[SW]
ANDNOT 754.05  ; 复测移载伺服X轴#1取料位[SW]
ANDNOT 754.06  ; 复测移载伺服X轴#2取料位[SW]
ANDNOT 754.07  ; 复测移载伺服X轴#1配对位[SW]
ANDNOT 754.08  ; 复测移载伺服X轴#2配对位[SW]
ANDNOT 754.09  ; 复测移载伺服X轴NG放料位[SW]
NOT(520)
ANDNOT P_On
AND W1.00  ; 手动模式
AND 755.15  ; 复测移载伺服Z轴跟踪开选择[SW]
ANDNOT 855.03  ; 复测移载伺服Z轴待机位标志[0055.03]
ANDNOT D1203.00  ; 复测移载机构：单步/自动循环运行中（总）
@SET 755.03  ; 复测移载伺服Z轴待机位[SW]

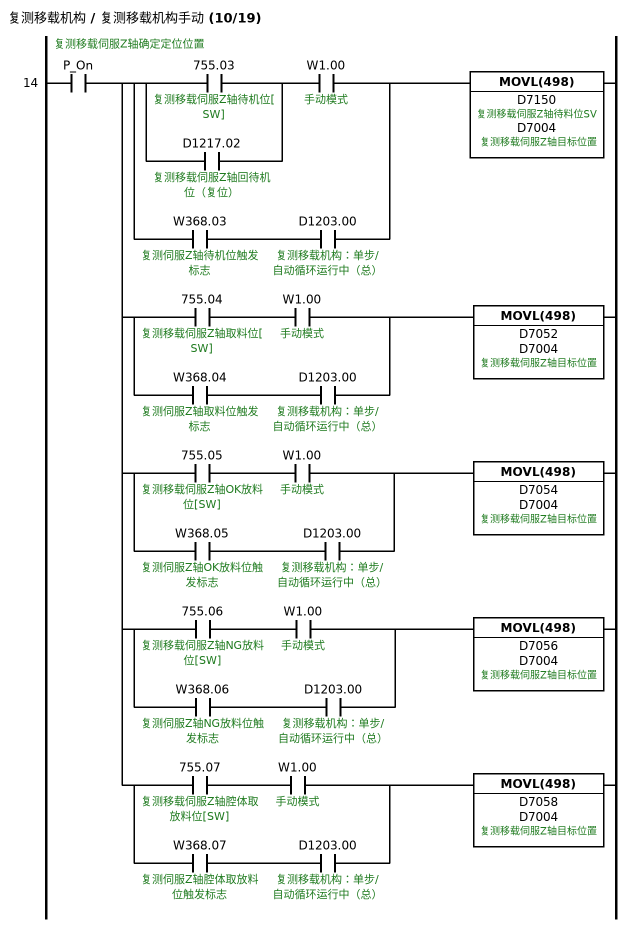
; rung 14: 复测移载伺服Z轴确定定位位置
LD P_On
OUT TR0
LD 755.03  ; 复测移载伺服Z轴待机位[SW]
OR D1217.02  ; 复测移载伺服Z轴回待机位（复位）
AND W1.00  ; 手动模式
LD W368.03  ; 复测伺服Z轴待机位触发标志
AND D1203.00  ; 复测移载机构：单步/自动循环运行中（总）
ORLD
ANDLD
MOVL(498) D7150 D7004  ; 复测移载伺服Z轴待料位SV, 复测移载伺服Z轴目标位置
LD TR0
LD 755.04  ; 复测移载伺服Z轴取料位[SW]
AND W1.00  ; 手动模式
LD W368.04  ; 复测伺服Z轴取料位触发标志
AND D1203.00  ; 复测移载机构：单步/自动循环运行中（总）
ORLD
ANDLD
MOVL(498) D7052 D7004  ; 复测移载伺服Z轴目标位置
LD TR0
LD 755.05  ; 复测移载伺服Z轴OK放料位[SW]
AND W1.00  ; 手动模式
LD W368.05  ; 复测伺服Z轴OK放料位触发标志
AND D1203.00  ; 复测移载机构：单步/自动循环运行中（总）
ORLD
ANDLD
MOVL(498) D7054 D7004  ; 复测移载伺服Z轴目标位置
LD TR0
LD 755.06  ; 复测移载伺服Z轴NG放料位[SW]
AND W1.00  ; 手动模式
LD W368.06  ; 复测伺服Z轴NG放料位触发标志
AND D1203.00  ; 复测移载机构：单步/自动循环运行中（总）
ORLD
ANDLD
MOVL(498) D7056 D7004  ; 复测移载伺服Z轴目标位置
LD TR0
LD 755.07  ; 复测移载伺服Z轴腔体取放料位[SW]
AND W1.00  ; 手动模式
LD W368.07  ; 复测伺服Z轴腔体取放料位触发标志
AND D1203.00  ; 复测移载机构：单步/自动循环运行中（总）
ORLD
ANDLD
MOVL(498) D7058 D7004  ; 复测移载伺服Z轴目标位置

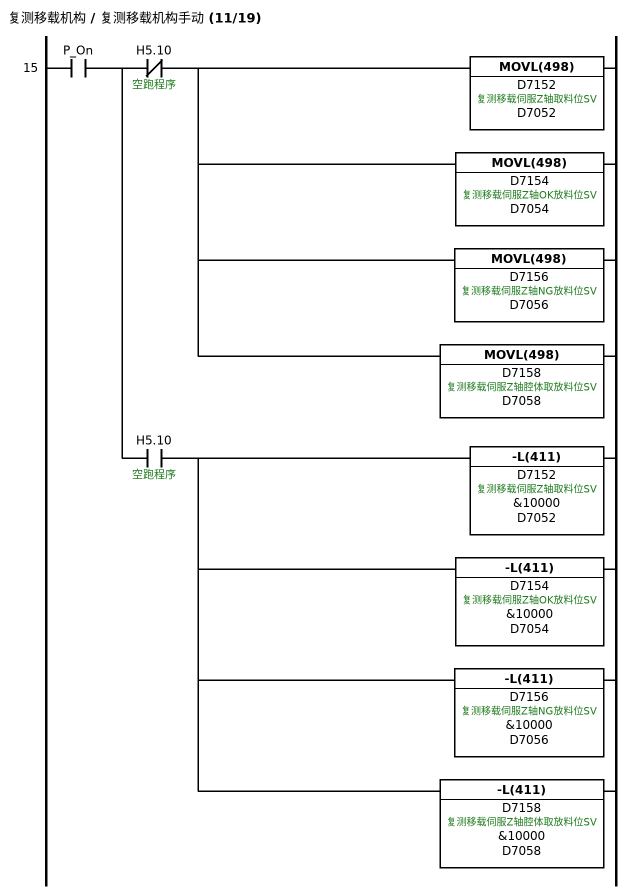
; rung 15
LD P_On
OUT TR0
ANDNOT H5.10  ; 空跑程序
MOVL(498) D7152 D7052  ; 复测移载伺服Z轴取料位SV
MOVL(498) D7154 D7054  ; 复测移载伺服Z轴OK放料位SV
MOVL(498) D7156 D7056  ; 复测移载伺服Z轴NG放料位SV
MOVL(498) D7158 D7058  ; 复测移载伺服Z轴腔体取放料位SV
LD TR0
AND H5.10  ; 空跑程序
-L(411) D7152 &10000 D7052  ; 复测移载伺服Z轴取料位SV
-L(411) D7154 &10000 D7054  ; 复测移载伺服Z轴OK放料位SV
-L(411) D7156 &10000 D7056  ; 复测移载伺服Z轴NG放料位SV
-L(411) D7158 &10000 D7058  ; 复测移载伺服Z轴腔体取放料位SV

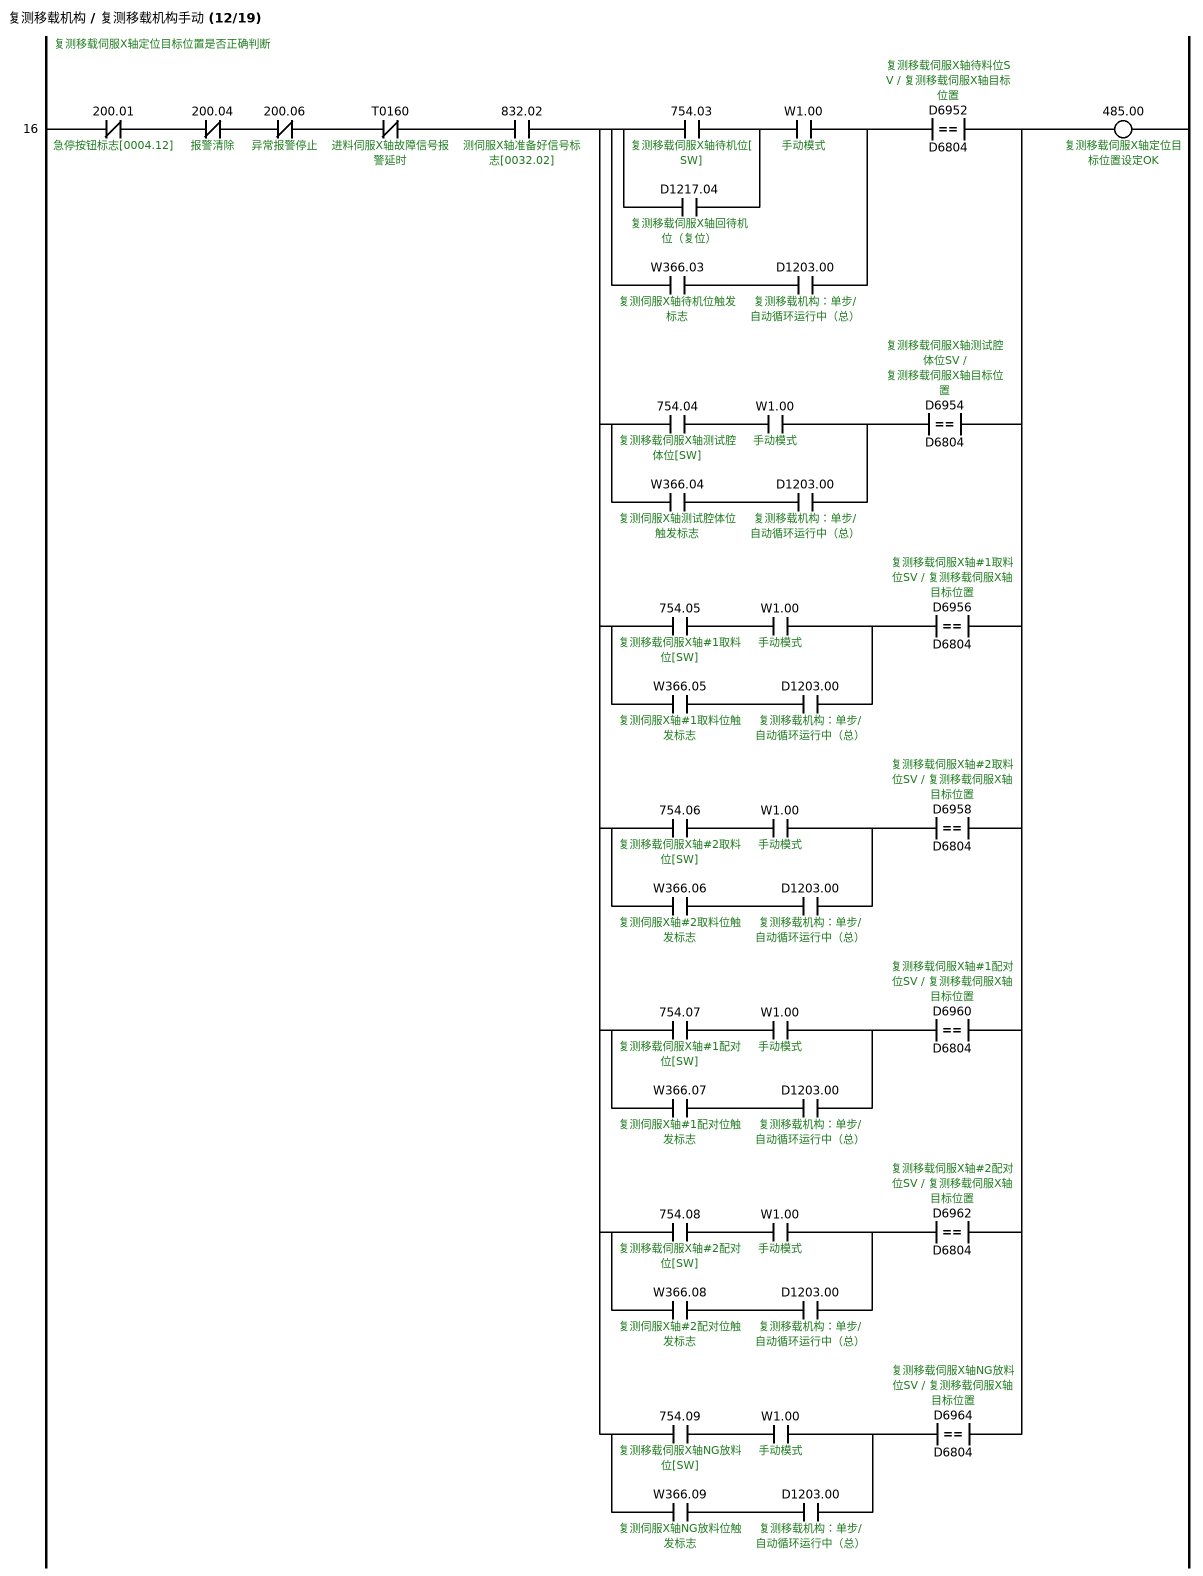
; rung 16: 复测移载伺服X轴定位目标位置是否正确判断
LDNOT 200.01  ; 急停按钮标志[0004.12]
ANDNOT 200.04  ; 报警清除
ANDNOT 200.06  ; 异常报警停止
ANDNOT T0160  ; 进料伺服X轴故障信号报警延时  // 待修改
AND 832.02  ; 测伺服X轴准备好信号标志[0032.02]
LD 754.03  ; 复测移载伺服X轴待机位[SW]
OR D1217.04  ; 复测移载伺服X轴回待机位（复位）
AND W1.00  ; 手动模式
LD W366.03  ; 复测伺服X轴待机位触发标志
AND D1203.00  ; 复测移载机构：单步/自动循环运行中（总）
ORLD
AND=SL(303) D6952 D6804  ; 复测移载伺服X轴待料位SV, 复测移载伺服X轴目标位置
LD 754.04  ; 复测移载伺服X轴测试腔体位[SW]
AND W1.00  ; 手动模式
LD W366.04  ; 复测伺服X轴测试腔体位触发标志
AND D1203.00  ; 复测移载机构：单步/自动循环运行中（总）
ORLD
AND=SL(303) D6954 D6804  ; 复测移载伺服X轴测试腔体位SV, 复测移载伺服X轴目标位置
ORLD
LD 754.05  ; 复测移载伺服X轴#1取料位[SW]
AND W1.00  ; 手动模式
LD W366.05  ; 复测伺服X轴#1取料位触发标志
AND D1203.00  ; 复测移载机构：单步/自动循环运行中（总）
ORLD
AND=SL(303) D6956 D6804  ; 复测移载伺服X轴#1取料位SV, 复测移载伺服X轴目标位置
ORLD
LD 754.06  ; 复测移载伺服X轴#2取料位[SW]
AND W1.00  ; 手动模式
LD W366.06  ; 复测伺服X轴#2取料位触发标志
AND D1203.00  ; 复测移载机构：单步/自动循环运行中（总）
ORLD
AND=SL(303) D6958 D6804  ; 复测移载伺服X轴#2取料位SV, 复测移载伺服X轴目标位置
ORLD
LD 754.07  ; 复测移载伺服X轴#1配对位[SW]
AND W1.00  ; 手动模式
LD W366.07  ; 复测伺服X轴#1配对位触发标志
AND D1203.00  ; 复测移载机构：单步/自动循环运行中（总）
ORLD
AND=SL(303) D6960 D6804  ; 复测移载伺服X轴#1配对位SV, 复测移载伺服X轴目标位置
ORLD
LD 754.08  ; 复测移载伺服X轴#2配对位[SW]
AND W1.00  ; 手动模式
LD W366.08  ; 复测伺服X轴#2配对位触发标志
AND D1203.00  ; 复测移载机构：单步/自动循环运行中（总）
ORLD
AND=SL(303) D6962 D6804  ; 复测移载伺服X轴#2配对位SV, 复测移载伺服X轴目标位置
ORLD
LD 754.09  ; 复测移载伺服X轴NG放料位[SW]
AND W1.00  ; 手动模式
LD W366.09  ; 复测伺服X轴NG放料位触发标志
AND D1203.00  ; 复测移载机构：单步/自动循环运行中（总）
ORLD
AND=SL(303) D6964 D6804  ; 复测移载伺服X轴NG放料位SV, 复测移载伺服X轴目标位置
ORLD
ANDLD
OUT 485.00  ; 复测移载伺服X轴定位目标位置设定OK

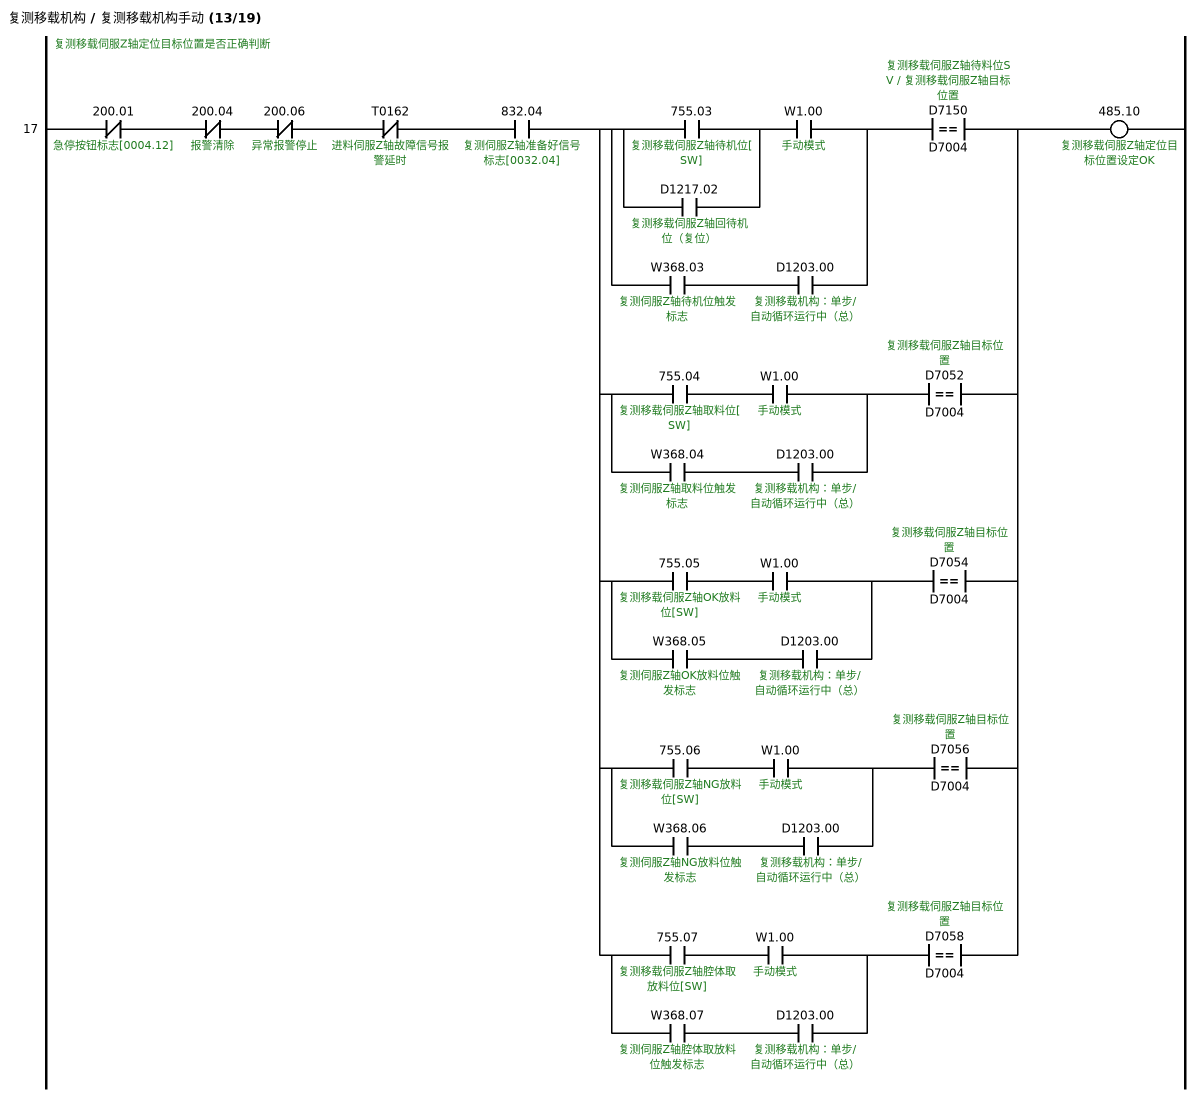
; rung 17: 复测移载伺服Z轴定位目标位置是否正确判断
LDNOT 200.01  ; 急停按钮标志[0004.12]
ANDNOT 200.04  ; 报警清除
ANDNOT 200.06  ; 异常报警停止
ANDNOT T0162  ; 进料伺服Z轴故障信号报警延时  // 待修改
AND 832.04  ; 复测伺服Z轴准备好信号标志[0032.04]
LD 755.03  ; 复测移载伺服Z轴待机位[SW]
OR D1217.02  ; 复测移载伺服Z轴回待机位（复位）
AND W1.00  ; 手动模式
LD W368.03  ; 复测伺服Z轴待机位触发标志
AND D1203.00  ; 复测移载机构：单步/自动循环运行中（总）
ORLD
AND=SL(303) D7150 D7004  ; 复测移载伺服Z轴待料位SV, 复测移载伺服Z轴目标位置
LD 755.04  ; 复测移载伺服Z轴取料位[SW]
AND W1.00  ; 手动模式
LD W368.04  ; 复测伺服Z轴取料位触发标志
AND D1203.00  ; 复测移载机构：单步/自动循环运行中（总）
ORLD
AND=SL(303) D7052 D7004  ; 复测移载伺服Z轴目标位置
ORLD
LD 755.05  ; 复测移载伺服Z轴OK放料位[SW]
AND W1.00  ; 手动模式
LD W368.05  ; 复测伺服Z轴OK放料位触发标志
AND D1203.00  ; 复测移载机构：单步/自动循环运行中（总）
ORLD
AND=SL(303) D7054 D7004  ; 复测移载伺服Z轴目标位置
ORLD
LD 755.06  ; 复测移载伺服Z轴NG放料位[SW]
AND W1.00  ; 手动模式
LD W368.06  ; 复测伺服Z轴NG放料位触发标志
AND D1203.00  ; 复测移载机构：单步/自动循环运行中（总）
ORLD
AND=SL(303) D7056 D7004  ; 复测移载伺服Z轴目标位置
ORLD
LD 755.07  ; 复测移载伺服Z轴腔体取放料位[SW]
AND W1.00  ; 手动模式
LD W368.07  ; 复测伺服Z轴腔体取放料位触发标志
AND D1203.00  ; 复测移载机构：单步/自动循环运行中（总）
ORLD
AND=SL(303) D7058 D7004  ; 复测移载伺服Z轴目标位置
ORLD
ANDLD
OUT 485.10  ; 复测移载伺服Z轴定位目标位置设定OK

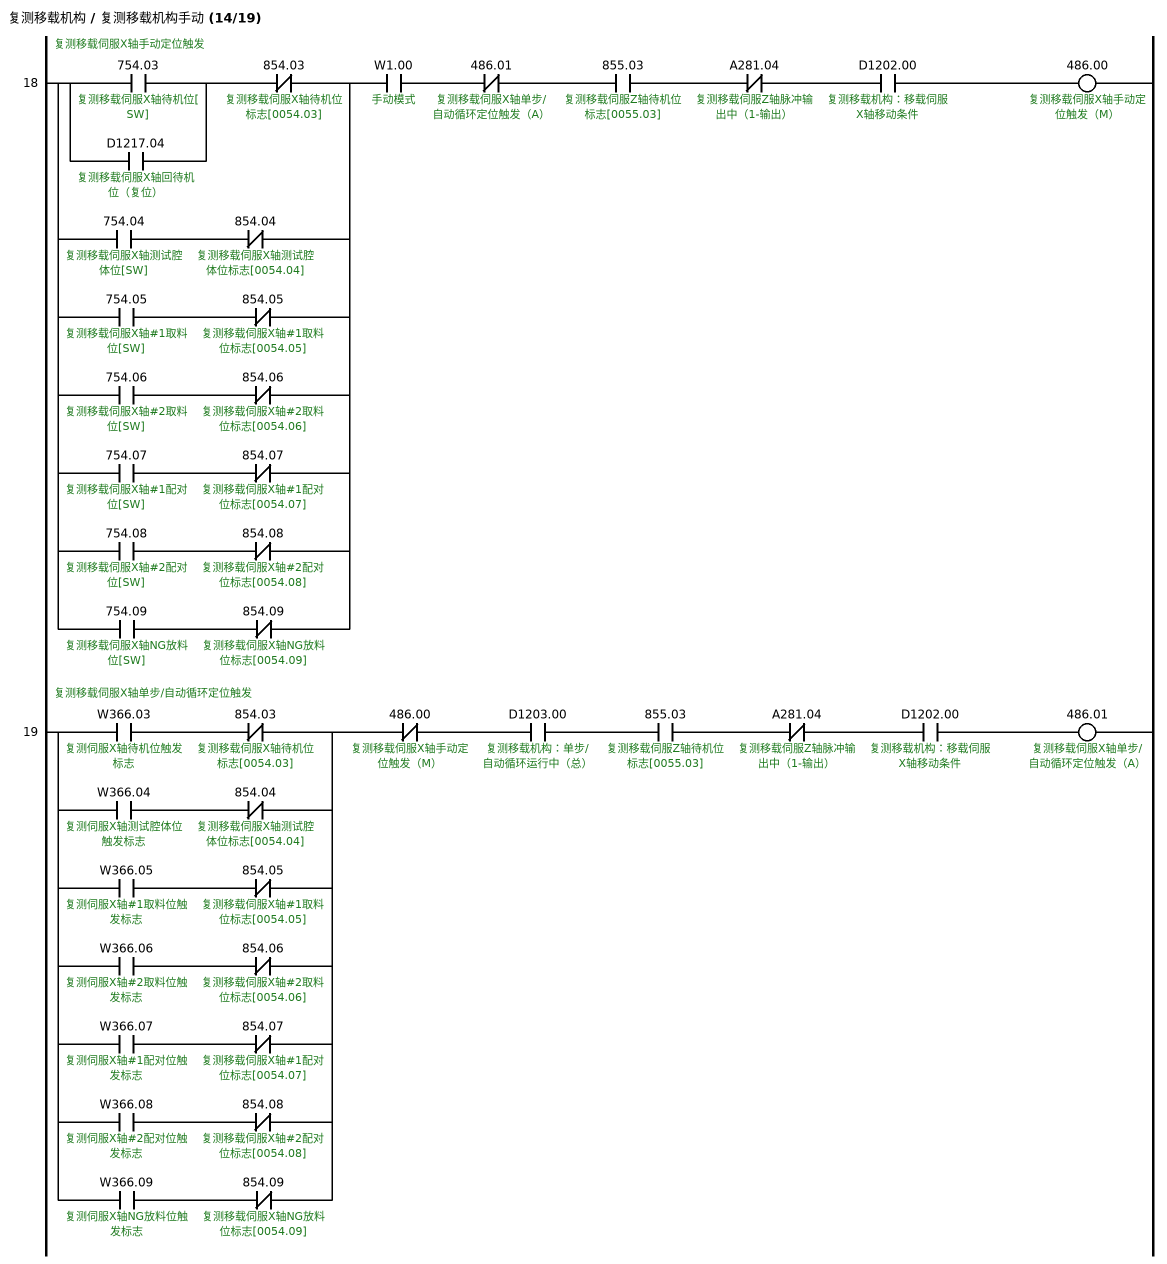
; rung 18: 复测移载伺服X轴手动定位触发
LD 754.03  ; 复测移载伺服X轴待机位[SW]
OR D1217.04  ; 复测移载伺服X轴回待机位（复位）
ANDNOT 854.03  ; 复测移载伺服X轴待机位标志[0054.03]
LD 754.04  ; 复测移载伺服X轴测试腔体位[SW]
ANDNOT 854.04  ; 复测移载伺服X轴测试腔体位标志[0054.04]
ORLD
LD 754.05  ; 复测移载伺服X轴#1取料位[SW]
ANDNOT 854.05  ; 复测移载伺服X轴#1取料位标志[0054.05]
ORLD
LD 754.06  ; 复测移载伺服X轴#2取料位[SW]
ANDNOT 854.06  ; 复测移载伺服X轴#2取料位标志[0054.06]
ORLD
LD 754.07  ; 复测移载伺服X轴#1配对位[SW]
ANDNOT 854.07  ; 复测移载伺服X轴#1配对位标志[0054.07]
ORLD
LD 754.08  ; 复测移载伺服X轴#2配对位[SW]
ANDNOT 854.08  ; 复测移载伺服X轴#2配对位标志[0054.08]
ORLD
LD 754.09  ; 复测移载伺服X轴NG放料位[SW]
ANDNOT 854.09  ; 复测移载伺服X轴NG放料位标志[0054.09]
ORLD
AND W1.00  ; 手动模式
ANDNOT 486.01  ; 复测移载伺服X轴单步/自动循环定位触发（A）
AND 855.03  ; 复测移载伺服Z轴待机位标志[0055.03]
ANDNOT A281.04  ; 复测移载伺服Z轴脉冲输出中（1-输出）
AND D1202.00  ; 复测移载机构：移载伺服X轴移动条件
OUT 486.00  ; 复测移载伺服X轴手动定位触发（M）
; rung 19: 复测移载伺服X轴单步/自动循环定位触发
LD W366.03  ; 复测伺服X轴待机位触发标志
ANDNOT 854.03  ; 复测移载伺服X轴待机位标志[0054.03]
LD W366.04  ; 复测伺服X轴测试腔体位触发标志
ANDNOT 854.04  ; 复测移载伺服X轴测试腔体位标志[0054.04]
ORLD
LD W366.05  ; 复测伺服X轴#1取料位触发标志
ANDNOT 854.05  ; 复测移载伺服X轴#1取料位标志[0054.05]
ORLD
LD W366.06  ; 复测伺服X轴#2取料位触发标志
ANDNOT 854.06  ; 复测移载伺服X轴#2取料位标志[0054.06]
ORLD
LD W366.07  ; 复测伺服X轴#1配对位触发标志
ANDNOT 854.07  ; 复测移载伺服X轴#1配对位标志[0054.07]
ORLD
LD W366.08  ; 复测伺服X轴#2配对位触发标志
ANDNOT 854.08  ; 复测移载伺服X轴#2配对位标志[0054.08]
ORLD
LD W366.09  ; 复测伺服X轴NG放料位触发标志
ANDNOT 854.09  ; 复测移载伺服X轴NG放料位标志[0054.09]
ORLD
ANDNOT 486.00  ; 复测移载伺服X轴手动定位触发（M）
AND D1203.00  ; 复测移载机构：单步/自动循环运行中（总）
AND 855.03  ; 复测移载伺服Z轴待机位标志[0055.03]
ANDNOT A281.04  ; 复测移载伺服Z轴脉冲输出中（1-输出）
AND D1202.00  ; 复测移载机构：移载伺服X轴移动条件
OUT 486.01  ; 复测移载伺服X轴单步/自动循环定位触发（A）

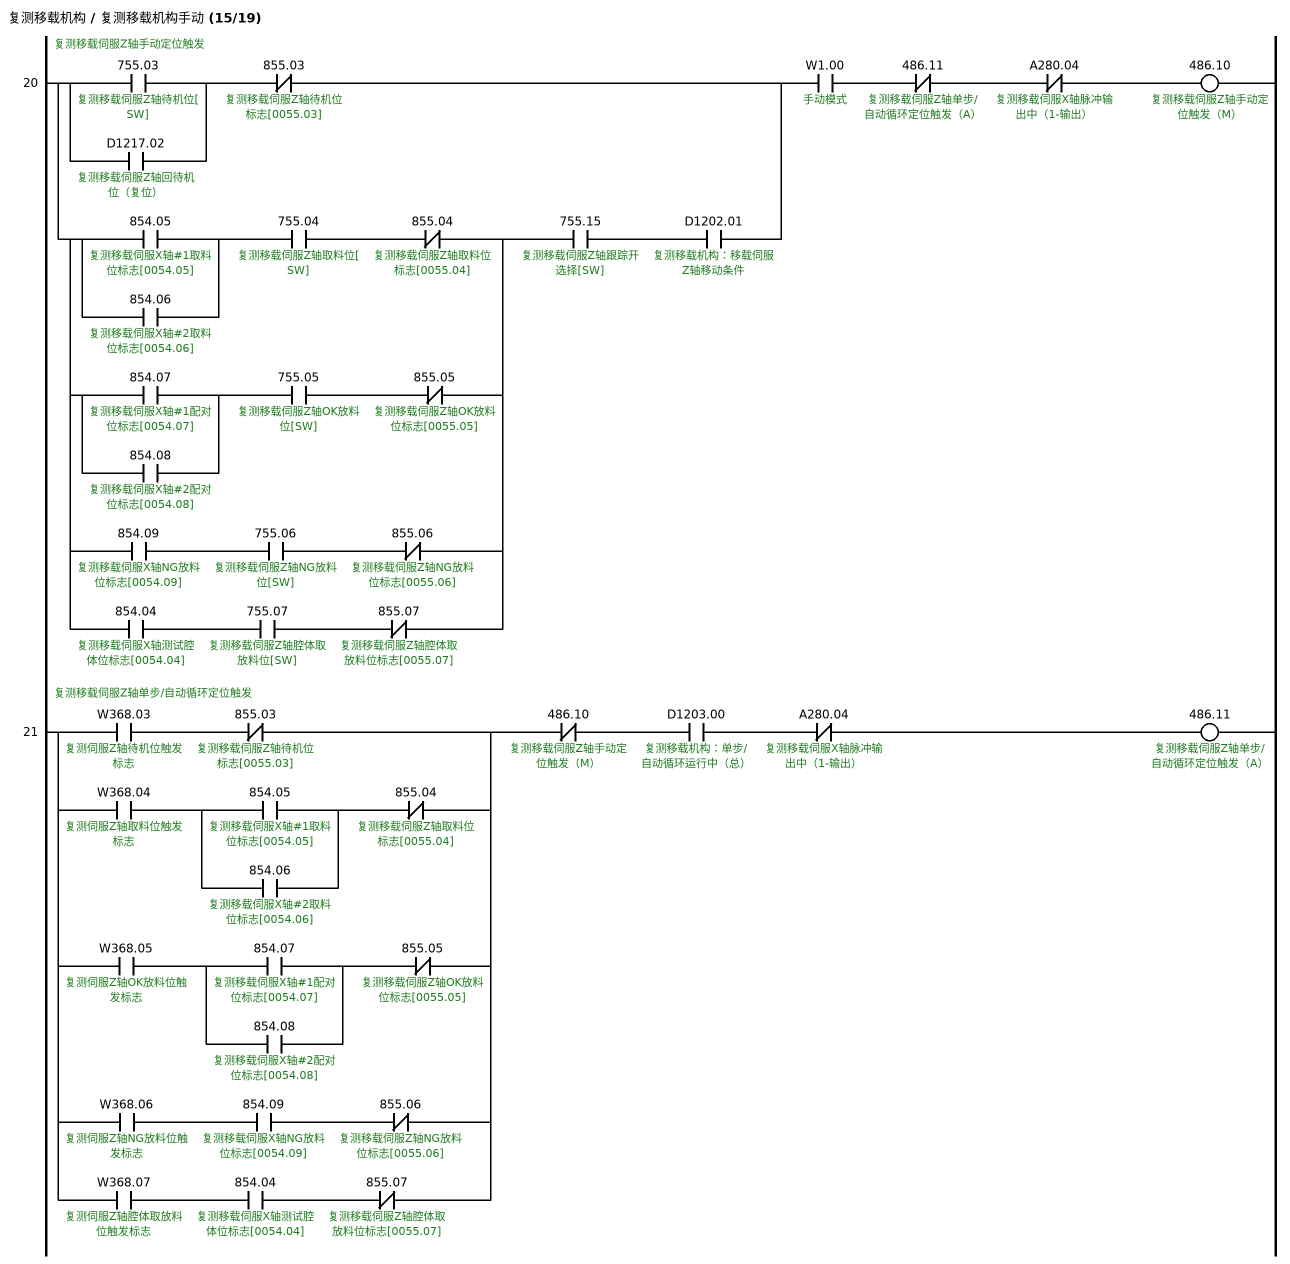
; rung 20: 复测移载伺服Z轴手动定位触发
LD 755.03  ; 复测移载伺服Z轴待机位[SW]
OR D1217.02  ; 复测移载伺服Z轴回待机位（复位）
ANDNOT 855.03  ; 复测移载伺服Z轴待机位标志[0055.03]
LD 854.05  ; 复测移载伺服X轴#1取料位标志[0054.05]
OR 854.06  ; 复测移载伺服X轴#2取料位标志[0054.06]
AND 755.04  ; 复测移载伺服Z轴取料位[SW]
ANDNOT 855.04  ; 复测移载伺服Z轴取料位标志[0055.04]
LD 854.07  ; 复测移载伺服X轴#1配对位标志[0054.07]
OR 854.08  ; 复测移载伺服X轴#2配对位标志[0054.08]
AND 755.05  ; 复测移载伺服Z轴OK放料位[SW]
ANDNOT 855.05  ; 复测移载伺服Z轴OK放料位标志[0055.05]
ORLD
LD 854.09  ; 复测移载伺服X轴NG放料位标志[0054.09]
AND 755.06  ; 复测移载伺服Z轴NG放料位[SW]
ANDNOT 855.06  ; 复测移载伺服Z轴NG放料位标志[0055.06]
ORLD
LD 854.04  ; 复测移载伺服X轴测试腔体位标志[0054.04]
AND 755.07  ; 复测移载伺服Z轴腔体取放料位[SW]
ANDNOT 855.07  ; 复测移载伺服Z轴腔体取放料位标志[0055.07]
ORLD
AND 755.15  ; 复测移载伺服Z轴跟踪开选择[SW]
AND D1202.01  ; 复测移载机构：移载伺服Z轴移动条件
ORLD
AND W1.00  ; 手动模式
ANDNOT 486.11  ; 复测移载伺服Z轴单步/自动循环定位触发（A）
ANDNOT A280.04  ; 复测移载伺服X轴脉冲输出中（1-输出）
OUT 486.10  ; 复测移载伺服Z轴手动定位触发（M）
; rung 21: 复测移载伺服Z轴单步/自动循环定位触发
LD W368.03  ; 复测伺服Z轴待机位触发标志
ANDNOT 855.03  ; 复测移载伺服Z轴待机位标志[0055.03]
LD W368.04  ; 复测伺服Z轴取料位触发标志
LD 854.05  ; 复测移载伺服X轴#1取料位标志[0054.05]
OR 854.06  ; 复测移载伺服X轴#2取料位标志[0054.06]
ANDLD
ANDNOT 855.04  ; 复测移载伺服Z轴取料位标志[0055.04]
ORLD
LD W368.05  ; 复测伺服Z轴OK放料位触发标志
LD 854.07  ; 复测移载伺服X轴#1配对位标志[0054.07]
OR 854.08  ; 复测移载伺服X轴#2配对位标志[0054.08]
ANDLD
ANDNOT 855.05  ; 复测移载伺服Z轴OK放料位标志[0055.05]
ORLD
LD W368.06  ; 复测伺服Z轴NG放料位触发标志
AND 854.09  ; 复测移载伺服X轴NG放料位标志[0054.09]
ANDNOT 855.06  ; 复测移载伺服Z轴NG放料位标志[0055.06]
ORLD
LD W368.07  ; 复测伺服Z轴腔体取放料位触发标志
AND 854.04  ; 复测移载伺服X轴测试腔体位标志[0054.04]
ANDNOT 855.07  ; 复测移载伺服Z轴腔体取放料位标志[0055.07]
ORLD
ANDNOT 486.10  ; 复测移载伺服Z轴手动定位触发（M）
AND D1203.00  ; 复测移载机构：单步/自动循环运行中（总）
ANDNOT A280.04  ; 复测移载伺服X轴脉冲输出中（1-输出）
OUT 486.11  ; 复测移载伺服Z轴单步/自动循环定位触发（A）

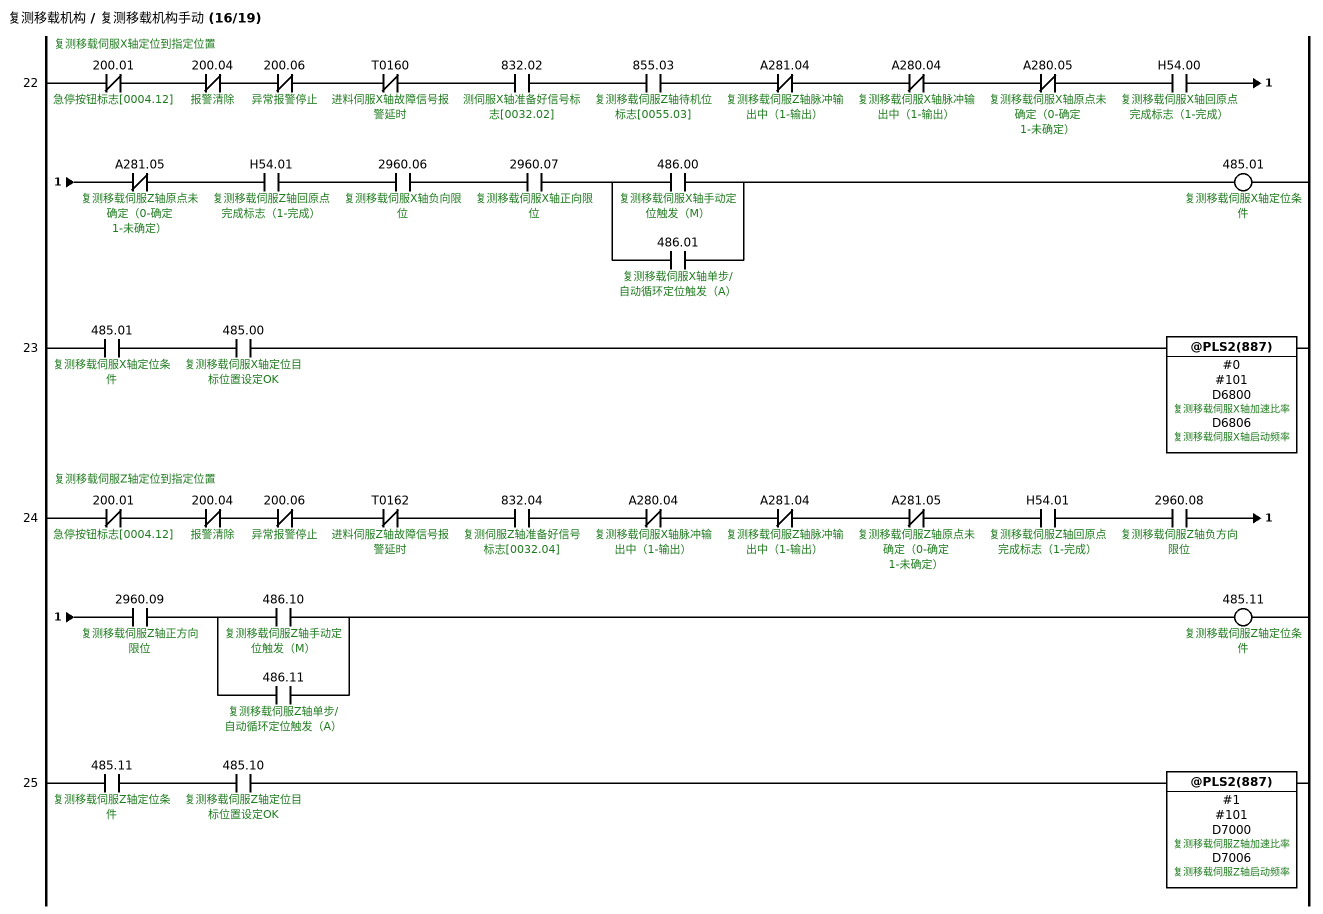
; rung 22: 复测移载伺服X轴定位到指定位置
LDNOT 200.01  ; 急停按钮标志[0004.12]
ANDNOT 200.04  ; 报警清除
ANDNOT 200.06  ; 异常报警停止
ANDNOT T0160  ; 进料伺服X轴故障信号报警延时  // 待修改
AND 832.02  ; 测伺服X轴准备好信号标志[0032.02]
AND 855.03  ; 复测移载伺服Z轴待机位标志[0055.03]
ANDNOT A281.04  ; 复测移载伺服Z轴脉冲输出中（1-输出）
ANDNOT A280.04  ; 复测移载伺服X轴脉冲输出中（1-输出）
ANDNOT A280.05  ; 复测移载伺服X轴原点未确定（0-确定  1-未确定）
AND H54.00  ; 复测移载伺服X轴回原点完成标志（1-完成）
ANDNOT A281.05  ; 复测移载伺服Z轴原点未确定（0-确定  1-未确定）
AND H54.01  ; 复测移载伺服Z轴回原点完成标志（1-完成）
AND 2960.06  ; 复测移载伺服X轴负向限位
AND 2960.07  ; 复测移载伺服X轴正向限位
LD 486.00  ; 复测移载伺服X轴手动定位触发（M）
OR 486.01  ; 复测移载伺服X轴单步/自动循环定位触发（A）
ANDLD
OUT 485.01  ; 复测移载伺服X轴定位条件
; rung 23
LD 485.01  ; 复测移载伺服X轴定位条件
AND 485.00  ; 复测移载伺服X轴定位目标位置设定OK
@PLS2(887) #0 #101 D6800 D6806  ; 复测移载伺服X轴加速比率, 复测移载伺服X轴启动频率
; rung 24: 复测移载伺服Z轴定位到指定位置
LDNOT 200.01  ; 急停按钮标志[0004.12]
ANDNOT 200.04  ; 报警清除
ANDNOT 200.06  ; 异常报警停止
ANDNOT T0162  ; 进料伺服Z轴故障信号报警延时  // 待修改
AND 832.04  ; 复测伺服Z轴准备好信号标志[0032.04]
ANDNOT A280.04  ; 复测移载伺服X轴脉冲输出中（1-输出）
ANDNOT A281.04  ; 复测移载伺服Z轴脉冲输出中（1-输出）
ANDNOT A281.05  ; 复测移载伺服Z轴原点未确定（0-确定  1-未确定）
AND H54.01  ; 复测移载伺服Z轴回原点完成标志（1-完成）
AND 2960.08  ; 复测移载伺服Z轴负方向限位
AND 2960.09  ; 复测移载伺服Z轴正方向限位
LD 486.10  ; 复测移载伺服Z轴手动定位触发（M）
OR 486.11  ; 复测移载伺服Z轴单步/自动循环定位触发（A）
ANDLD
OUT 485.11  ; 复测移载伺服Z轴定位条件
; rung 25
LD 485.11  ; 复测移载伺服Z轴定位条件
AND 485.10  ; 复测移载伺服Z轴定位目标位置设定OK
@PLS2(887) #1 #101 D7000 D7006  ; 复测移载伺服Z轴加速比率, 复测移载伺服Z轴启动频率

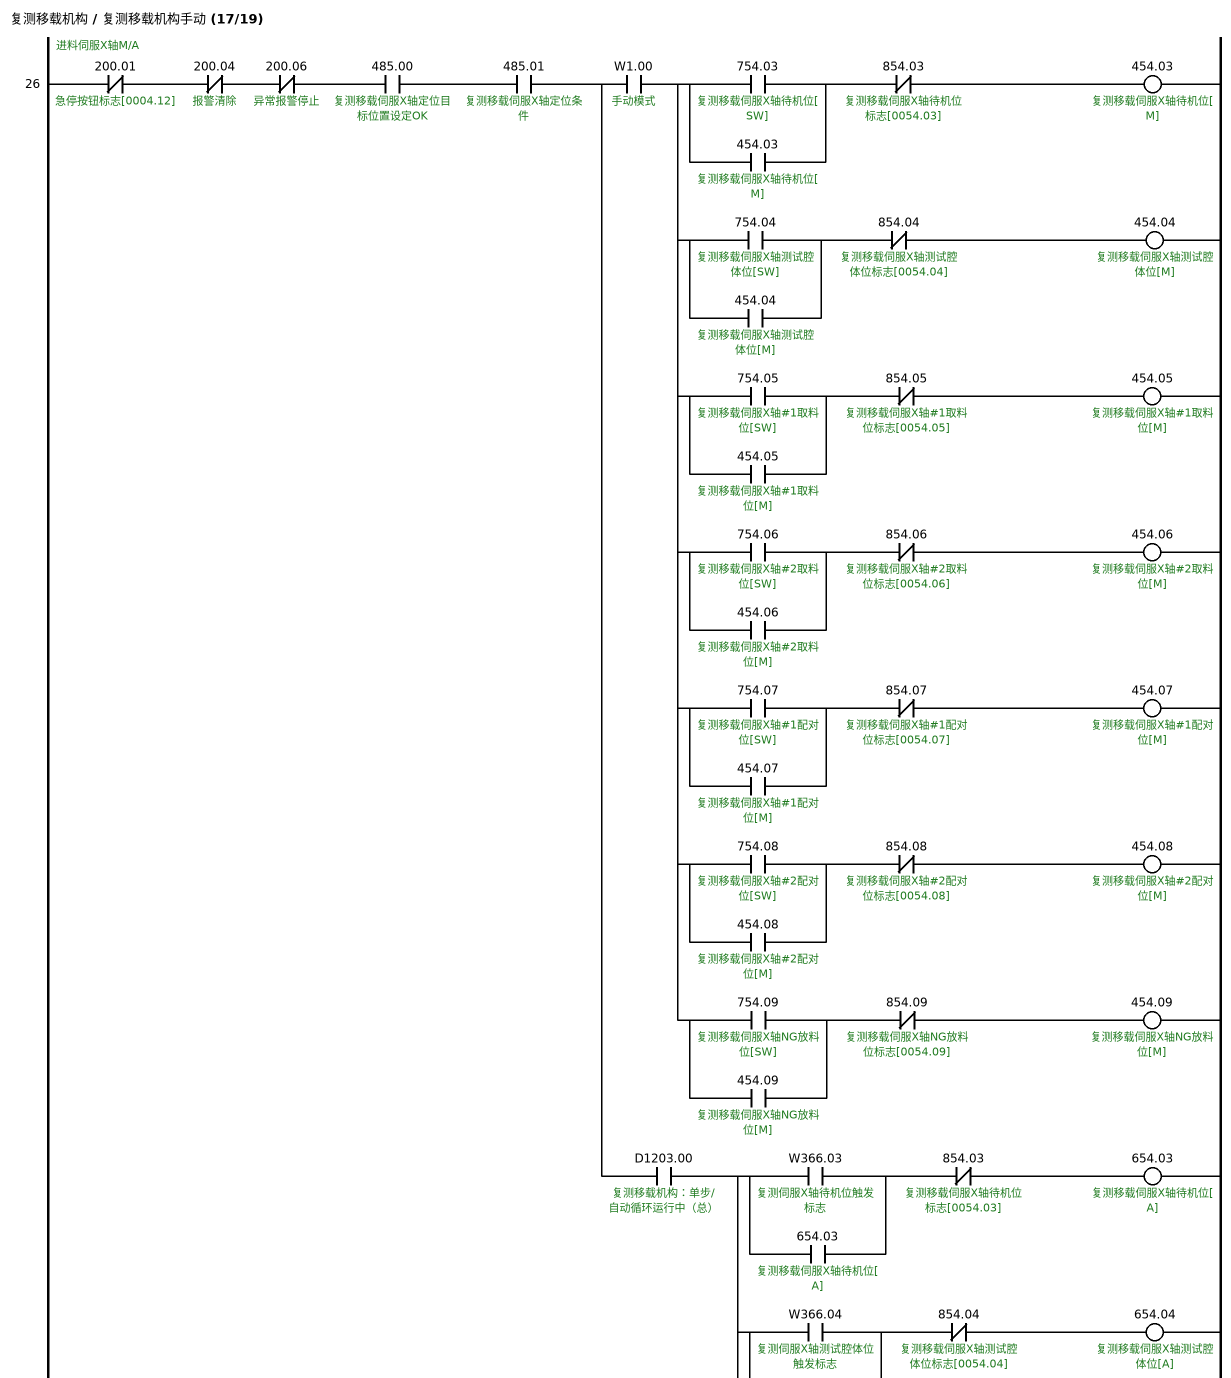

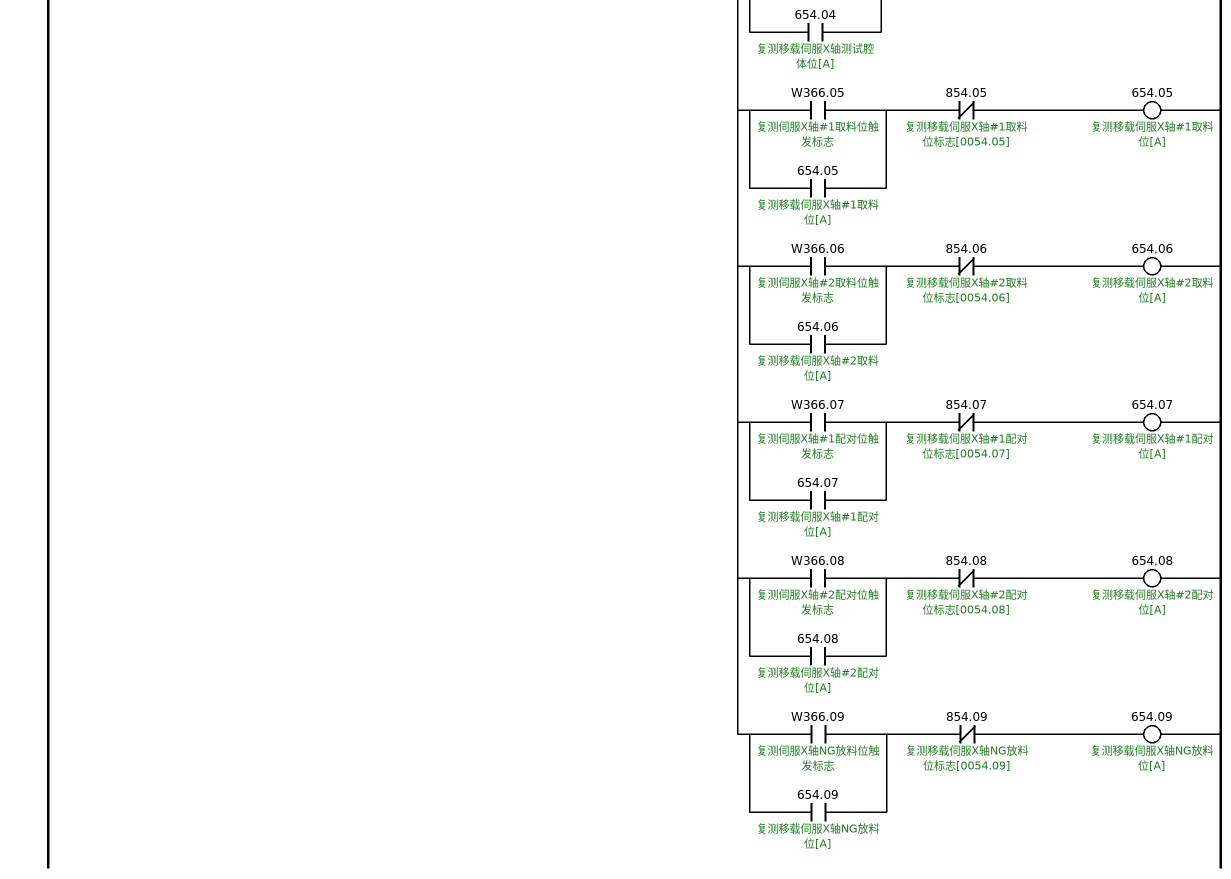
; rung 26: 进料伺服X轴M/A
LDNOT 200.01  ; 急停按钮标志[0004.12]
ANDNOT 200.04  ; 报警清除
ANDNOT 200.06  ; 异常报警停止
AND 485.00  ; 复测移载伺服X轴定位目标位置设定OK
AND 485.01  ; 复测移载伺服X轴定位条件
OUT TR0
AND W1.00  ; 手动模式
OUT TR1
LD 754.03  ; 复测移载伺服X轴待机位[SW]
OR 454.03  ; 复测移载伺服X轴待机位[M]
ANDLD
ANDNOT 854.03  ; 复测移载伺服X轴待机位标志[0054.03]
OUT 454.03  ; 复测移载伺服X轴待机位[M]
LD TR1
LD 754.04  ; 复测移载伺服X轴测试腔体位[SW]
OR 454.04  ; 复测移载伺服X轴测试腔体位[M]
ANDLD
ANDNOT 854.04  ; 复测移载伺服X轴测试腔体位标志[0054.04]
OUT 454.04  ; 复测移载伺服X轴测试腔体位[M]
LD TR1
LD 754.05  ; 复测移载伺服X轴#1取料位[SW]
OR 454.05  ; 复测移载伺服X轴#1取料位[M]
ANDLD
ANDNOT 854.05  ; 复测移载伺服X轴#1取料位标志[0054.05]
OUT 454.05  ; 复测移载伺服X轴#1取料位[M]
LD TR1
LD 754.06  ; 复测移载伺服X轴#2取料位[SW]
OR 454.06  ; 复测移载伺服X轴#2取料位[M]
ANDLD
ANDNOT 854.06  ; 复测移载伺服X轴#2取料位标志[0054.06]
OUT 454.06  ; 复测移载伺服X轴#2取料位[M]
LD TR1
LD 754.07  ; 复测移载伺服X轴#1配对位[SW]
OR 454.07  ; 复测移载伺服X轴#1配对位[M]
ANDLD
ANDNOT 854.07  ; 复测移载伺服X轴#1配对位标志[0054.07]
OUT 454.07  ; 复测移载伺服X轴#1配对位[M]
LD TR1
LD 754.08  ; 复测移载伺服X轴#2配对位[SW]
OR 454.08  ; 复测移载伺服X轴#2配对位[M]
ANDLD
ANDNOT 854.08  ; 复测移载伺服X轴#2配对位标志[0054.08]
OUT 454.08  ; 复测移载伺服X轴#2配对位[M]
LD TR1
LD 754.09  ; 复测移载伺服X轴NG放料位[SW]
OR 454.09  ; 复测移载伺服X轴NG放料位[M]
ANDLD
ANDNOT 854.09  ; 复测移载伺服X轴NG放料位标志[0054.09]
OUT 454.09  ; 复测移载伺服X轴NG放料位[M]
LD TR0
AND D1203.00  ; 复测移载机构：单步/自动循环运行中（总）
OUT TR0
LD W366.03  ; 复测伺服X轴待机位触发标志
OR 654.03  ; 复测移载伺服X轴待机位[A]
ANDLD
ANDNOT 854.03  ; 复测移载伺服X轴待机位标志[0054.03]
OUT 654.03  ; 复测移载伺服X轴待机位[A]
LD TR0
LD W366.04  ; 复测伺服X轴测试腔体位触发标志
OR 654.04  ; 复测移载伺服X轴测试腔体位[A]
ANDLD
ANDNOT 854.04  ; 复测移载伺服X轴测试腔体位标志[0054.04]
OUT 654.04  ; 复测移载伺服X轴测试腔体位[A]
LD TR0
LD W366.05  ; 复测伺服X轴#1取料位触发标志
OR 654.05  ; 复测移载伺服X轴#1取料位[A]
ANDLD
ANDNOT 854.05  ; 复测移载伺服X轴#1取料位标志[0054.05]
OUT 654.05  ; 复测移载伺服X轴#1取料位[A]
LD TR0
LD W366.06  ; 复测伺服X轴#2取料位触发标志
OR 654.06  ; 复测移载伺服X轴#2取料位[A]
ANDLD
ANDNOT 854.06  ; 复测移载伺服X轴#2取料位标志[0054.06]
OUT 654.06  ; 复测移载伺服X轴#2取料位[A]
LD TR0
LD W366.07  ; 复测伺服X轴#1配对位触发标志
OR 654.07  ; 复测移载伺服X轴#1配对位[A]
ANDLD
ANDNOT 854.07  ; 复测移载伺服X轴#1配对位标志[0054.07]
OUT 654.07  ; 复测移载伺服X轴#1配对位[A]
LD TR0
LD W366.08  ; 复测伺服X轴#2配对位触发标志
OR 654.08  ; 复测移载伺服X轴#2配对位[A]
ANDLD
ANDNOT 854.08  ; 复测移载伺服X轴#2配对位标志[0054.08]
OUT 654.08  ; 复测移载伺服X轴#2配对位[A]
LD TR0
LD W366.09  ; 复测伺服X轴NG放料位触发标志
OR 654.09  ; 复测移载伺服X轴NG放料位[A]
ANDLD
ANDNOT 854.09  ; 复测移载伺服X轴NG放料位标志[0054.09]
OUT 654.09  ; 复测移载伺服X轴NG放料位[A]

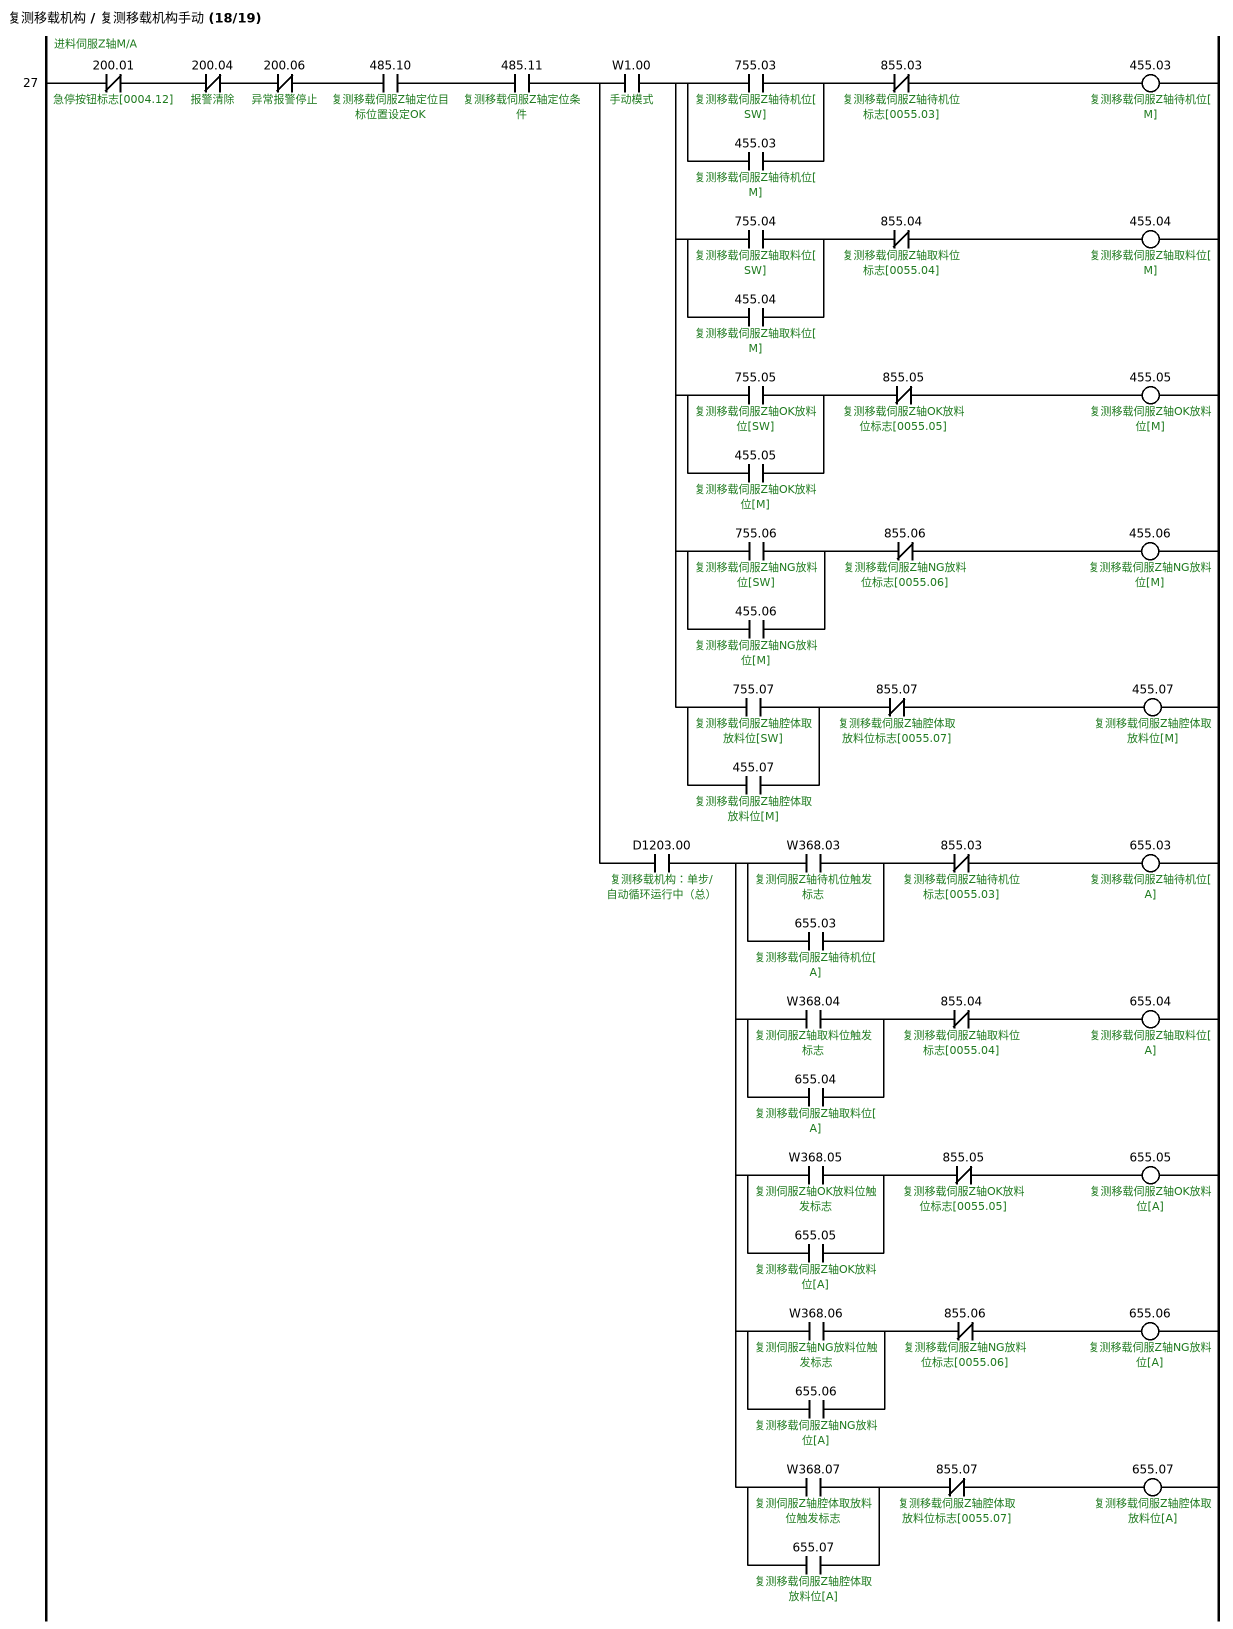
; rung 27: 进料伺服Z轴M/A
LDNOT 200.01  ; 急停按钮标志[0004.12]
ANDNOT 200.04  ; 报警清除
ANDNOT 200.06  ; 异常报警停止
AND 485.10  ; 复测移载伺服Z轴定位目标位置设定OK
AND 485.11  ; 复测移载伺服Z轴定位条件
OUT TR0
AND W1.00  ; 手动模式
OUT TR1
LD 755.03  ; 复测移载伺服Z轴待机位[SW]
OR 455.03  ; 复测移载伺服Z轴待机位[M]
ANDLD
ANDNOT 855.03  ; 复测移载伺服Z轴待机位标志[0055.03]
OUT 455.03  ; 复测移载伺服Z轴待机位[M]
LD TR1
LD 755.04  ; 复测移载伺服Z轴取料位[SW]
OR 455.04  ; 复测移载伺服Z轴取料位[M]
ANDLD
ANDNOT 855.04  ; 复测移载伺服Z轴取料位标志[0055.04]
OUT 455.04  ; 复测移载伺服Z轴取料位[M]
LD TR1
LD 755.05  ; 复测移载伺服Z轴OK放料位[SW]
OR 455.05  ; 复测移载伺服Z轴OK放料位[M]
ANDLD
ANDNOT 855.05  ; 复测移载伺服Z轴OK放料位标志[0055.05]
OUT 455.05  ; 复测移载伺服Z轴OK放料位[M]
LD TR1
LD 755.06  ; 复测移载伺服Z轴NG放料位[SW]
OR 455.06  ; 复测移载伺服Z轴NG放料位[M]
ANDLD
ANDNOT 855.06  ; 复测移载伺服Z轴NG放料位标志[0055.06]
OUT 455.06  ; 复测移载伺服Z轴NG放料位[M]
LD TR1
LD 755.07  ; 复测移载伺服Z轴腔体取放料位[SW]
OR 455.07  ; 复测移载伺服Z轴腔体取放料位[M]
ANDLD
ANDNOT 855.07  ; 复测移载伺服Z轴腔体取放料位标志[0055.07]
OUT 455.07  ; 复测移载伺服Z轴腔体取放料位[M]
LD TR0
AND D1203.00  ; 复测移载机构：单步/自动循环运行中（总）
OUT TR0
LD W368.03  ; 复测伺服Z轴待机位触发标志
OR 655.03  ; 复测移载伺服Z轴待机位[A]
ANDLD
ANDNOT 855.03  ; 复测移载伺服Z轴待机位标志[0055.03]
OUT 655.03  ; 复测移载伺服Z轴待机位[A]
LD TR0
LD W368.04  ; 复测伺服Z轴取料位触发标志
OR 655.04  ; 复测移载伺服Z轴取料位[A]
ANDLD
ANDNOT 855.04  ; 复测移载伺服Z轴取料位标志[0055.04]
OUT 655.04  ; 复测移载伺服Z轴取料位[A]
LD TR0
LD W368.05  ; 复测伺服Z轴OK放料位触发标志
OR 655.05  ; 复测移载伺服Z轴OK放料位[A]
ANDLD
ANDNOT 855.05  ; 复测移载伺服Z轴OK放料位标志[0055.05]
OUT 655.05  ; 复测移载伺服Z轴OK放料位[A]
LD TR0
LD W368.06  ; 复测伺服Z轴NG放料位触发标志
OR 655.06  ; 复测移载伺服Z轴NG放料位[A]
ANDLD
ANDNOT 855.06  ; 复测移载伺服Z轴NG放料位标志[0055.06]
OUT 655.06  ; 复测移载伺服Z轴NG放料位[A]
LD TR0
LD W368.07  ; 复测伺服Z轴腔体取放料位触发标志
OR 655.07  ; 复测移载伺服Z轴腔体取放料位[A]
ANDLD
ANDNOT 855.07  ; 复测移载伺服Z轴腔体取放料位标志[0055.07]
OUT 655.07  ; 复测移载伺服Z轴腔体取放料位[A]

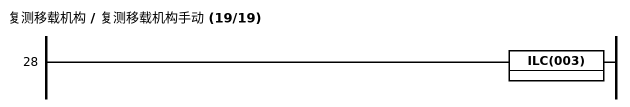
; rung 28
ILC(003)

### Section 工站复位

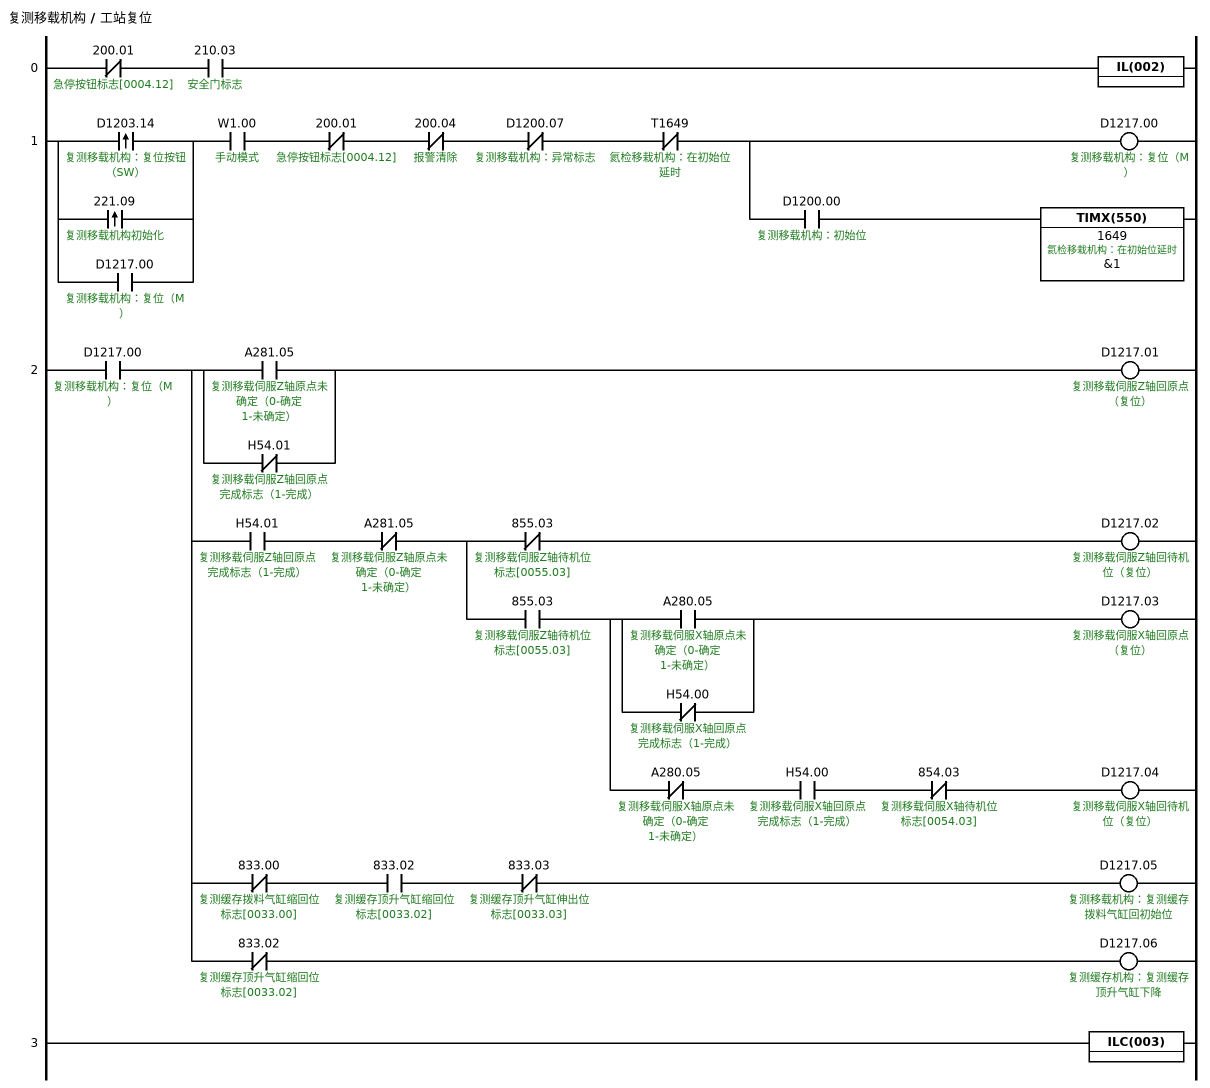
; rung 0
LDNOT 200.01  ; 急停按钮标志[0004.12]
AND 210.03  ; 安全门标志
IL(002)
; rung 1
@LD D1203.14  ; 复测移载机构：复位按钮（SW）
@OR 221.09  ; 复测移载机构初始化
OR D1217.00  ; 复测移载机构：复位（M）
AND W1.00  ; 手动模式
ANDNOT 200.01  ; 急停按钮标志[0004.12]
ANDNOT 200.04  ; 报警清除
ANDNOT D1200.07  ; 复测移载机构：异常标志
ANDNOT T1649  ; 氦检移栽机构：在初始位延时
OUT D1217.00  ; 复测移载机构：复位（M）
AND D1200.00  ; 复测移载机构：初始位
TIMX(550) 1649 &1  ; 氦检移栽机构：在初始位延时
; rung 2
LD D1217.00  ; 复测移载机构：复位（M）
OUT TR0
LD A281.05  ; 复测移载伺服Z轴原点未确定（0-确定  1-未确定）
ORNOT H54.01  ; 复测移载伺服Z轴回原点完成标志（1-完成）
ANDLD
OUT D1217.01  ; 复测移载伺服Z轴回原点（复位）
LD TR0
AND H54.01  ; 复测移载伺服Z轴回原点完成标志（1-完成）
ANDNOT A281.05  ; 复测移载伺服Z轴原点未确定（0-确定  1-未确定）
OUT TR1
ANDNOT 855.03  ; 复测移载伺服Z轴待机位标志[0055.03]
OUT D1217.02  ; 复测移载伺服Z轴回待机位（复位）
LD TR1
AND 855.03  ; 复测移载伺服Z轴待机位标志[0055.03]
OUT TR1
LD A280.05  ; 复测移载伺服X轴原点未确定（0-确定  1-未确定）
ORNOT H54.00  ; 复测移载伺服X轴回原点完成标志（1-完成）
ANDLD
OUT D1217.03  ; 复测移载伺服X轴回原点（复位）
LD TR1
ANDNOT A280.05  ; 复测移载伺服X轴原点未确定（0-确定  1-未确定）
AND H54.00  ; 复测移载伺服X轴回原点完成标志（1-完成）
ANDNOT 854.03  ; 复测移载伺服X轴待机位标志[0054.03]
OUT D1217.04  ; 复测移载伺服X轴回待机位（复位）
LD TR0
ANDNOT 833.00  ; 复测缓存拨料气缸缩回位标志[0033.00]
AND 833.02  ; 复测缓存顶升气缸缩回位标志[0033.02]
ANDNOT 833.03  ; 复测缓存顶升气缸伸出位标志[0033.03]
OUT D1217.05  ; 复测移载机构：复测缓存拨料气缸回初始位
LD TR0
ANDNOT 833.02  ; 复测缓存顶升气缸缩回位标志[0033.02]
OUT D1217.06  ; 复测缓存机构：复测缓存顶升气缸下降
; rung 3
ILC(003)

### Section 指示灯

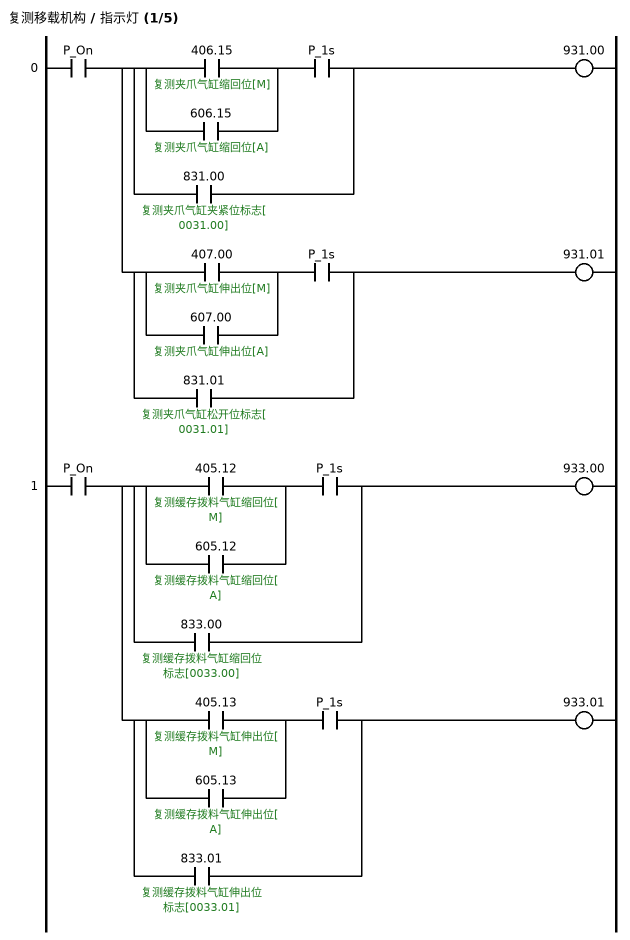
; rung 0
LD P_On
OUT TR0
LD 406.15  ; 复测夹爪气缸缩回位[M]
OR 606.15  ; 复测夹爪气缸缩回位[A]
AND P_1s
OR 831.00  ; 复测夹爪气缸夹紧位标志[0031.00]
ANDLD
OUT 931.00
LD TR0
LD 407.00  ; 复测夹爪气缸伸出位[M]
OR 607.00  ; 复测夹爪气缸伸出位[A]
AND P_1s
OR 831.01  ; 复测夹爪气缸松开位标志[0031.01]
ANDLD
OUT 931.01
; rung 1
LD P_On
OUT TR0
LD 405.12  ; 复测缓存拨料气缸缩回位[M]
OR 605.12  ; 复测缓存拨料气缸缩回位[A]
AND P_1s
OR 833.00  ; 复测缓存拨料气缸缩回位标志[0033.00]
ANDLD
OUT 933.00
LD TR0
LD 405.13  ; 复测缓存拨料气缸伸出位[M]
OR 605.13  ; 复测缓存拨料气缸伸出位[A]
AND P_1s
OR 833.01  ; 复测缓存拨料气缸伸出位标志[0033.01]
ANDLD
OUT 933.01

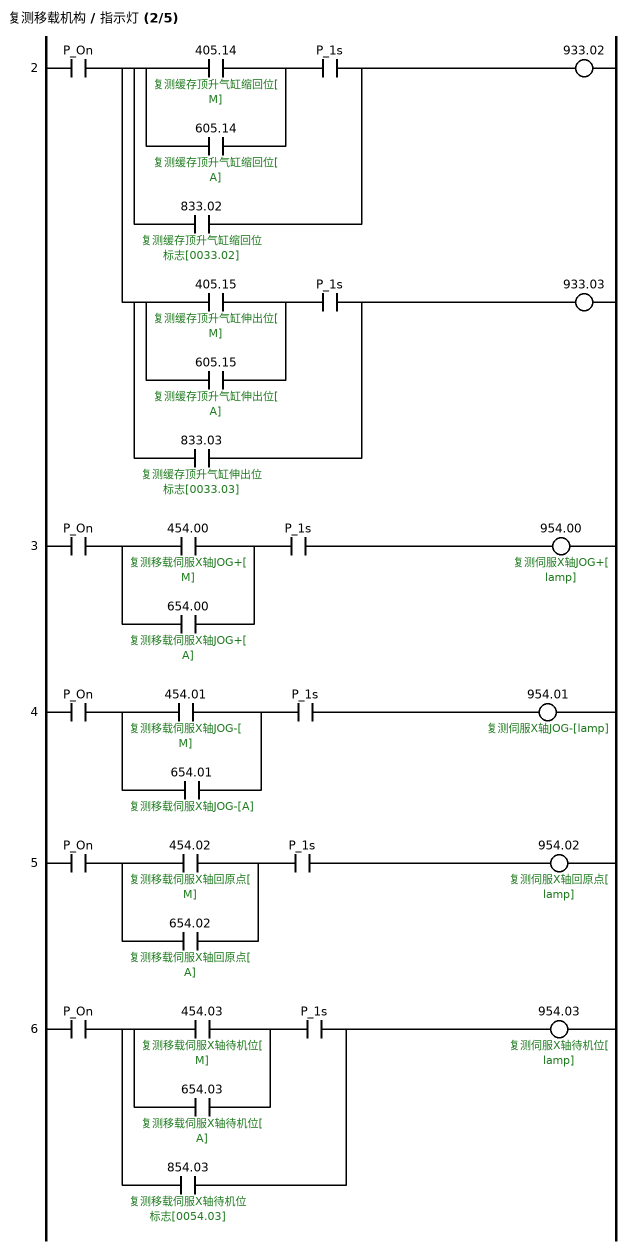
; rung 2
LD P_On
OUT TR0
LD 405.14  ; 复测缓存顶升气缸缩回位[M]
OR 605.14  ; 复测缓存顶升气缸缩回位[A]
AND P_1s
OR 833.02  ; 复测缓存顶升气缸缩回位标志[0033.02]
ANDLD
OUT 933.02
LD TR0
LD 405.15  ; 复测缓存顶升气缸伸出位[M]
OR 605.15  ; 复测缓存顶升气缸伸出位[A]
AND P_1s
OR 833.03  ; 复测缓存顶升气缸伸出位标志[0033.03]
ANDLD
OUT 933.03
; rung 3
LD P_On
LD 454.00  ; 复测移载伺服X轴JOG+[M]
OR 654.00  ; 复测移载伺服X轴JOG+[A]
ANDLD
AND P_1s
OUT 954.00  ; 复测伺服X轴JOG+[lamp]
; rung 4
LD P_On
LD 454.01  ; 复测移载伺服X轴JOG-[M]
OR 654.01  ; 复测移载伺服X轴JOG-[A]
ANDLD
AND P_1s
OUT 954.01  ; 复测伺服X轴JOG-[lamp]
; rung 5
LD P_On
LD 454.02  ; 复测移载伺服X轴回原点[M]
OR 654.02  ; 复测移载伺服X轴回原点[A]
ANDLD
AND P_1s
OUT 954.02  ; 复测伺服X轴回原点[lamp]
; rung 6
LD P_On
LD 454.03  ; 复测移载伺服X轴待机位[M]
OR 654.03  ; 复测移载伺服X轴待机位[A]
AND P_1s
OR 854.03  ; 复测移载伺服X轴待机位标志[0054.03]
ANDLD
OUT 954.03  ; 复测伺服X轴待机位[lamp]

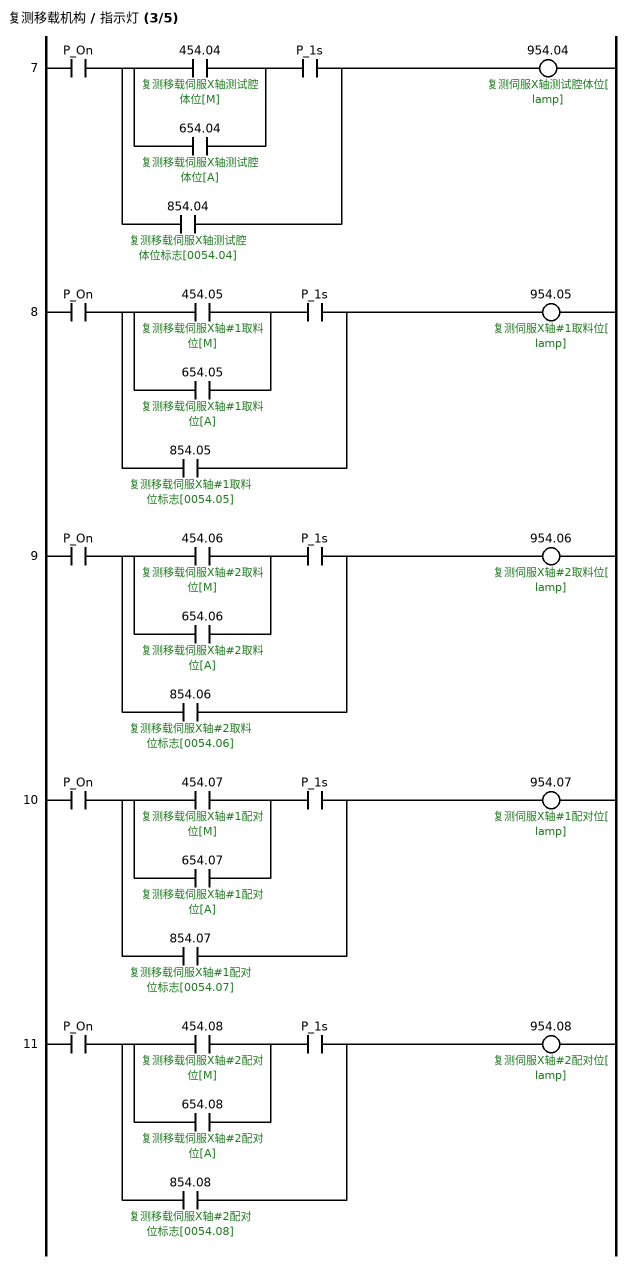
; rung 7
LD P_On
LD 454.04  ; 复测移载伺服X轴测试腔体位[M]
OR 654.04  ; 复测移载伺服X轴测试腔体位[A]
AND P_1s
OR 854.04  ; 复测移载伺服X轴测试腔体位标志[0054.04]
ANDLD
OUT 954.04  ; 复测伺服X轴测试腔体位[lamp]
; rung 8
LD P_On
LD 454.05  ; 复测移载伺服X轴#1取料位[M]
OR 654.05  ; 复测移载伺服X轴#1取料位[A]
AND P_1s
OR 854.05  ; 复测移载伺服X轴#1取料位标志[0054.05]
ANDLD
OUT 954.05  ; 复测伺服X轴#1取料位[lamp]
; rung 9
LD P_On
LD 454.06  ; 复测移载伺服X轴#2取料位[M]
OR 654.06  ; 复测移载伺服X轴#2取料位[A]
AND P_1s
OR 854.06  ; 复测移载伺服X轴#2取料位标志[0054.06]
ANDLD
OUT 954.06  ; 复测伺服X轴#2取料位[lamp]
; rung 10
LD P_On
LD 454.07  ; 复测移载伺服X轴#1配对位[M]
OR 654.07  ; 复测移载伺服X轴#1配对位[A]
AND P_1s
OR 854.07  ; 复测移载伺服X轴#1配对位标志[0054.07]
ANDLD
OUT 954.07  ; 复测伺服X轴#1配对位[lamp]
; rung 11
LD P_On
LD 454.08  ; 复测移载伺服X轴#2配对位[M]
OR 654.08  ; 复测移载伺服X轴#2配对位[A]
AND P_1s
OR 854.08  ; 复测移载伺服X轴#2配对位标志[0054.08]
ANDLD
OUT 954.08  ; 复测伺服X轴#2配对位[lamp]

